LIN {X 0,Y 524.655,Z 657.487,A -85,B 0,C 180,E1 -4783.755,E2 -4783.755} C_VEL
LIN {X 0,Y 525.074,Z 645.522,A -85,B 0,C 180,E1 -4784.931,E2 -4784.931} C_VEL
LIN {X 0,Y 525.538,Z 633.607,A -85,B 0,C 180,E1 -4785.91,E2 -4785.91} C_VEL
LIN {X 0,Y 525.983,Z 620.728,A -85,B 0,C 180,E1 -4786.794,E2 -4786.794} C_VEL
LIN {X 0,Y 526.424,Z 606.681,A -85,B 0,C 180,E1 -4787.581,E2 -4787.581} C_VEL
LIN {X 0,Y 526.898,Z 592.222,A -85,B 0,C 180,E1 -4788.217,E2 -4788.217} C_VEL
LIN {X 0,Y 527.248,Z 577.139,A -85,B 0,C 180,E1 -4788.715,E2 -4788.715} C_VEL
LIN {X 0,Y 527.506,Z 562.381,A -85,B 0,C 180,E1 -4789.05,E2 -4789.05} C_VEL
LIN {X 0,Y 528.507,Z 412.087,A -85,B 0,C 180,E1 -4791.163,E2 -4791.163} C_VEL
LIN {X 0,Y 525.9,Z 396.895,A -85,B 0,C 180,E1 -4791.514,E2 -4791.514} C_VEL
LIN {X 0,Y 526.479,Z 374.491,A -85,B 0,C 180,E1 -4794.235,E2 -4794.235} C_VEL
LIN {X 0,Y 527.196,Z 352.396,A -85,B 0,C 180,E1 -4796.952,E2 -4796.952} C_VEL
LIN {X 0,Y 527.268,Z 349.014,A -85,B 0,C 180,E1 -4797.377,E2 -4797.377} C_VEL
LIN {X 0,Y 524.306,Z 336.37,A -85,B 0,C 180,E1 -4799.154,E2 -4799.154} C_VEL
LIN {X 0,Y 523.938,Z 334.849,A -85,B 0,C 180,E1 -4799.406,E2 -4799.406} C_VEL
LIN {X 0,Y 523.931,Z 334.844,A -85,B 0,C 180,E1 -4802.449,E2 -4802.449} C_VEL
LIN {X 0,Y 523.918,Z 334.851,A -85,B 0,C 180,E1 -4805.226,E2 -4805.226} C_VEL
LIN {X 0,Y 523.914,Z 334.848,A -85,B 0,C 180,E1 -4808.101,E2 -4808.101} C_VEL
LIN {X 0,Y 523.96,Z 334.847,A -85,B 0,C 180,E1 -4811.311,E2 -4811.311} C_VEL
LIN {X 0,Y 523.954,Z 334.841,A -85,B 0,C 180,E1 -4814.691,E2 -4814.691} C_VEL
LIN {X 0,Y 523.954,Z 334.84,A -85,B 0,C 180,E1 -4817.881,E2 -4817.881} C_VEL
LIN {X 0,Y 523.919,Z 334.848,A -85,B 0,C 180,E1 -4820.915,E2 -4820.915} C_VEL
LIN {X 0,Y 523.925,Z 334.843,A -85,B 0,C 180,E1 -4823.828,E2 -4823.828} C_VEL
LIN {X 0,Y 523.939,Z 334.843,A -85,B 0,C 180,E1 -4826.636,E2 -4826.636} C_VEL
LIN {X 0,Y 523.952,Z 334.844,A -85,B 0,C 180,E1 -4829.356,E2 -4829.356} C_VEL
LIN {X 0,Y 523.974,Z 334.836,A -85,B 0,C 180,E1 -4832.281,E2 -4832.281} C_VEL
LIN {X 0,Y 523.95,Z 334.841,A -85,B 0,C 180,E1 -4834.581,E2 -4834.581} C_VEL
LIN {X 0,Y 523.914,Z 334.853,A -85,B 0,C 180,E1 -4837.107,E2 -4837.107} C_VEL
LIN {X 0,Y 523.976,Z 334.836,A -85,B 0,C 180,E1 -4839.866,E2 -4839.866} C_VEL
LIN {X 0,Y 523.964,Z 334.844,A -85,B 0,C 180,E1 -4842.837,E2 -4842.837} C_VEL
LIN {X 0,Y 523.974,Z 334.842,A -85,B 0,C 180,E1 -4845.236,E2 -4845.236} C_VEL
LIN {X 0,Y 524.01,Z 334.833,A -85,B 0,C 180,E1 -4848.394,E2 -4848.394} C_VEL
LIN {X 0,Y 524.001,Z 334.835,A -85,B 0,C 180,E1 -4851.516,E2 -4851.516} C_VEL
LIN {X 0,Y 524.079,Z 334.827,A -85,B 0,C 180,E1 -4854.614,E2 -4854.614} C_VEL
LIN {X 0,Y 524.111,Z 334.82,A -85,B 0,C 180,E1 -4857.695,E2 -4857.695} C_VEL
LIN {X 0,Y 524.122,Z 334.825,A -85,B 0,C 180,E1 -4860.769,E2 -4860.769} C_VEL
LIN {X 0,Y 524.068,Z 334.831,A -85,B 0,C 180,E1 -4863.075,E2 -4863.075} C_VEL
LIN {X 0,Y 524.049,Z 334.828,A -85,B 0,C 180,E1 -4866.159,E2 -4866.159} C_VEL
LIN {X 0,Y 523.997,Z 334.836,A -85,B 0,C 180,E1 -4869.262,E2 -4869.262} C_VEL
LIN {X 0,Y 524.001,Z 334.833,A -85,B 0,C 180,E1 -4871.74,E2 -4871.74} C_VEL
LIN {X 0,Y 523.991,Z 334.839,A -85,B 0,C 180,E1 -4875.053,E2 -4875.053} C_VEL
LIN {X 0,Y 523.962,Z 334.838,A -85,B 0,C 180,E1 -4877.969,E2 -4877.969} C_VEL
LIN {X 0,Y 523.97,Z 334.841,A -85,B 0,C 180,E1 -4880.41,E2 -4880.41} C_VEL
LIN {X 0,Y 523.909,Z 334.851,A -85,B 0,C 180,E1 -4882.894,E2 -4882.894} C_VEL
LIN {X 0,Y 523.934,Z 334.842,A -85,B 0,C 180,E1 -4885.42,E2 -4885.42} C_VEL
LIN {X 0,Y 523.952,Z 334.84,A -85,B 0,C 180,E1 -4888,E2 -4888} C_VEL
LIN {X 0,Y 523.944,Z 334.847,A -85,B 0,C 180,E1 -4890.855,E2 -4890.855} C_VEL
LIN {X 0,Y 523.96,Z 334.838,A -85,B 0,C 180,E1 -4893.735,E2 -4893.735} C_VEL
LIN {X 0,Y 523.919,Z 334.849,A -85,B 0,C 180,E1 -4896.404,E2 -4896.404} C_VEL
LIN {X 0,Y 523.919,Z 334.846,A -85,B 0,C 180,E1 -4899.085,E2 -4899.085} C_VEL
LIN {X 0,Y 523.94,Z 334.843,A -85,B 0,C 180,E1 -4902.121,E2 -4902.121} C_VEL
LIN {X 0,Y 523.941,Z 334.841,A -85,B 0,C 180,E1 -4905.311,E2 -4905.311} C_VEL
LIN {X 0,Y 523.9,Z 334.849,A -85,B 0,C 180,E1 -4906.913,E2 -4906.913} C_VEL
LIN {X 0,Y 523.24,Z 334.929,A -85,B 0,C 180,E1 -4907.555,E2 -4907.555} C_VEL
LIN {X 0,Y 520.406,Z 335.29,A -85,B 0,C 180,E1 -4908.597,E2 -4908.597} C_VEL
LIN {X 0,Y 518.005,Z 335.589,A -85,B 0,C 180,E1 -4909.436,E2 -4909.436} C_VEL
LIN {X 0,Y 516.969,Z 335.715,A -85,B 0,C 180,E1 -4910.083,E2 -4910.083} C_VEL
LIN {X 0,Y 516.882,Z 335.725,A -85,B 0,C 180,E1 -4910.303,E2 -4910.303} C_VEL
LIN {X 0,Y 516.854,Z 335.723,A -85,B 0,C 180,E1 -4913.347,E2 -4913.347} C_VEL
LIN {X 0,Y 516.908,Z 335.72,A -85,B 0,C 180,E1 -4916.121,E2 -4916.121} C_VEL
LIN {X 0,Y 516.891,Z 335.721,A -85,B 0,C 180,E1 -4918.937,E2 -4918.937} C_VEL
LIN {X 0,Y 516.863,Z 335.722,A -85,B 0,C 180,E1 -4921.582,E2 -4921.582} C_VEL
LIN {X 0,Y 516.879,Z 335.725,A -85,B 0,C 180,E1 -4924.209,E2 -4924.209} C_VEL
LIN {X 0,Y 516.86,Z 335.726,A -85,B 0,C 180,E1 -4926.776,E2 -4926.776} C_VEL
LIN {X 0,Y 516.94,Z 335.713,A -85,B 0,C 180,E1 -4929.733,E2 -4929.733} C_VEL
LIN {X 0,Y 516.882,Z 335.726,A -85,B 0,C 180,E1 -4932.595,E2 -4932.595} C_VEL
LIN {X 0,Y 516.939,Z 335.714,A -85,B 0,C 180,E1 -4935.03,E2 -4935.03} C_VEL
LIN {X 0,Y 516.971,Z 335.716,A -85,B 0,C 180,E1 -4938.234,E2 -4938.234} C_VEL
LIN {X 0,Y 516.934,Z 335.713,A -85,B 0,C 180,E1 -4941.399,E2 -4941.399} C_VEL
LIN {X 0,Y 516.985,Z 335.712,A -85,B 0,C 180,E1 -4944.54,E2 -4944.54} C_VEL
LIN {X 0,Y 517.077,Z 335.697,A -85,B 0,C 180,E1 -4947.663,E2 -4947.663} C_VEL
LIN {X 0,Y 517.01,Z 335.706,A -85,B 0,C 180,E1 -4950.779,E2 -4950.779} C_VEL
LIN {X 0,Y 517.076,Z 335.703,A -85,B 0,C 180,E1 -4952.337,E2 -4952.337} C_VEL
LIN {X 0,Y 516.975,Z 335.717,A -85,B 0,C 180,E1 -4956.244,E2 -4956.244} C_VEL
LIN {X 0,Y 516.911,Z 335.716,A -85,B 0,C 180,E1 -4959.39,E2 -4959.39} C_VEL
LIN {X 0,Y 516.902,Z 335.722,A -85,B 0,C 180,E1 -4962.565,E2 -4962.565} C_VEL
LIN {X 0,Y 516.832,Z 335.733,A -85,B 0,C 180,E1 -4965.782,E2 -4965.782} C_VEL
LIN {X 0,Y 516.878,Z 335.791,A -85,B 0,C 180,E1 -4967.049,E2 -4967.049} C_VEL
LIN {X 0,Y 518.301,Z 342.495,A -85,B 0,C 180,E1 -4968.249,E2 -4968.249} C_VEL
LIN {X 0,Y 520.55,Z 349.737,A -85,B 0,C 180,E1 -4968.46,E2 -4968.46} C_VEL
LIN {X 0,Y 521.981,Z 356.506,A -85,B 0,C 180,E1 -4968.624,E2 -4968.624} C_VEL
LIN {X 0,Y 520.841,Z 507.169,A -85,B 0,C 180,E1 -4970.79,E2 -4970.79} C_VEL
LIN {X 0,Y 520.577,Z 522.264,A -85,B 0,C 180,E1 -4971.165,E2 -4971.165} C_VEL
LIN {X 0,Y 520.179,Z 537.472,A -85,B 0,C 180,E1 -4971.707,E2 -4971.707} C_VEL
LIN {X 0,Y 519.763,Z 552.073,A -85,B 0,C 180,E1 -4972.403,E2 -4972.403} C_VEL
LIN {X 0,Y 519.251,Z 565.638,A -85,B 0,C 180,E1 -4973.217,E2 -4973.217} C_VEL
LIN {X 0,Y 518.701,Z 578.837,A -85,B 0,C 180,E1 -4974.189,E2 -4974.189} C_VEL
LIN {X 0,Y 518.145,Z 591.198,A -85,B 0,C 180,E1 -4975.294,E2 -4975.294} C_VEL
LIN {X 0,Y 517.709,Z 601.985,A -85,B 0,C 180,E1 -4976.451,E2 -4976.451} C_VEL
LIN {X 0,Y 517.308,Z 612.091,A -85,B 0,C 180,E1 -4977.74,E2 -4977.74} C_VEL
LIN {X 0,Y 516.968,Z 620.889,A -85,B 0,C 180,E1 -4979.079,E2 -4979.079} C_VEL
LIN {X 0,Y 516.683,Z 629.217,A -85,B 0,C 180,E1 -4980.61,E2 -4980.61} C_VEL
LIN {X 0,Y 516.497,Z 635.604,A -85,B 0,C 180,E1 -4982.051,E2 -4982.051} C_VEL
LIN {X 0,Y 516.368,Z 640.556,A -85,B 0,C 180,E1 -4983.426,E2 -4983.426} C_VEL
LIN {X 0,Y 516.253,Z 644.668,A -85,B 0,C 180,E1 -4984.874,E2 -4984.874} C_VEL
LIN {X 0,Y 516.177,Z 648.074,A -85,B 0,C 180,E1 -4986.552,E2 -4986.552} C_VEL
LIN {X 0,Y 516.14,Z 649.735,A -85,B 0,C 180,E1 -4987.837,E2 -4987.837} C_VEL
LIN {X 0,Y 516.152,Z 650.678,A -85,B 0,C 180,E1 -4989.093,E2 -4989.093} C_VEL
LIN {X 0,Y 516.173,Z 650.75,A -85,B 0,C 180,E1 -4990.81,E2 -4990.81} C_VEL
LIN {X 0,Y 516.166,Z 650.148,A -85,B 0,C 180,E1 -4991.85,E2 -4991.85} C_VEL
LIN {X 0,Y 516.175,Z 648.994,A -85,B 0,C 180,E1 -4992.905,E2 -4992.905} C_VEL
LIN {X 0,Y 516.288,Z 646.397,A -85,B 0,C 180,E1 -4994.453,E2 -4994.453} C_VEL
LIN {X 0,Y 516.383,Z 642.122,A -85,B 0,C 180,E1 -4996.165,E2 -4996.165} C_VEL
LIN {X 0,Y 516.442,Z 636.865,A -85,B 0,C 180,E1 -4997.735,E2 -4997.735} C_VEL
LIN {X 0,Y 516.635,Z 630.492,A -85,B 0,C 180,E1 -4999.234,E2 -4999.234} C_VEL
LIN {X 0,Y 516.904,Z 622.228,A -85,B 0,C 180,E1 -5000.805,E2 -5000.805} C_VEL
LIN {X 0,Y 517.25,Z 613.537,A -85,B 0,C 180,E1 -5002.161,E2 -5002.161} C_VEL
LIN {X 0,Y 517.705,Z 602.748,A -85,B 0,C 180,E1 -5003.564,E2 -5003.564} C_VEL
LIN {X 0,Y 518.226,Z 591.212,A -85,B 0,C 180,E1 -5004.804,E2 -5004.804} C_VEL
LIN {X 0,Y 518.709,Z 578.953,A -85,B 0,C 180,E1 -5005.902,E2 -5005.902} C_VEL
LIN {X 0,Y 519.183,Z 566.64,A -85,B 0,C 180,E1 -5006.818,E2 -5006.818} C_VEL
LIN {X 0,Y 519.754,Z 552.758,A -85,B 0,C 180,E1 -5007.659,E2 -5007.659} C_VEL
LIN {X 0,Y 520.167,Z 538.55,A -85,B 0,C 180,E1 -5008.342,E2 -5008.342} C_VEL
LIN {X 0,Y 520.558,Z 522.971,A -85,B 0,C 180,E1 -5008.908,E2 -5008.908} C_VEL
LIN {X 0,Y 520.81,Z 507.957,A -85,B 0,C 180,E1 -5009.285,E2 -5009.285} C_VEL
LIN {X 0,Y 521.407,Z 427.366,A -85,B 0,C 180,E1 -5010.459,E2 -5010.459} C_VEL
LIN {X 0,Y 521.907,Z 355.675,A -85,B 0,C 180,E1 -5011.489,E2 -5011.489} C_VEL
LIN {X 0,Y 519.249,Z 345.342,A -85,B 0,C 180,E1 -5011.761,E2 -5011.761} C_VEL
LIN {X 0,Y 518.421,Z 342.909,A -85,B 0,C 180,E1 -5011.862,E2 -5011.862} C_VEL
LIN {X 0,Y 516.883,Z 335.728,A -85,B 0,C 180,E1 -5013.203,E2 -5013.203} C_VEL
LIN {X 0,Y 516.871,Z 335.729,A -85,B 0,C 180,E1 -5015.926,E2 -5015.926} C_VEL
LIN {X 0,Y 516.867,Z 335.724,A -85,B 0,C 180,E1 -5018.461,E2 -5018.461} C_VEL
LIN {X 0,Y 516.882,Z 335.721,A -85,B 0,C 180,E1 -5020.954,E2 -5020.954} C_VEL
LIN {X 0,Y 516.844,Z 335.728,A -85,B 0,C 180,E1 -5023.408,E2 -5023.408} C_VEL
LIN {X 0,Y 516.884,Z 335.728,A -85,B 0,C 180,E1 -5025.833,E2 -5025.833} C_VEL
LIN {X 0,Y 516.95,Z 335.714,A -85,B 0,C 180,E1 -5029.028,E2 -5029.028} C_VEL
LIN {X 0,Y 516.926,Z 335.717,A -85,B 0,C 180,E1 -5032.186,E2 -5032.186} C_VEL
LIN {X 0,Y 516.989,Z 335.707,A -85,B 0,C 180,E1 -5034.539,E2 -5034.539} C_VEL
LIN {X 0,Y 517.078,Z 335.704,A -85,B 0,C 180,E1 -5037.663,E2 -5037.663} C_VEL
LIN {X 0,Y 517.088,Z 335.698,A -85,B 0,C 180,E1 -5040,E2 -5040} C_VEL
LIN {X 0,Y 517.082,Z 335.696,A -85,B 0,C 180,E1 -5042.337,E2 -5042.337} C_VEL
LIN {X 0,Y 517.015,Z 335.711,A -85,B 0,C 180,E1 -5045.46,E2 -5045.46} C_VEL
LIN {X 0,Y 516.957,Z 335.712,A -85,B 0,C 180,E1 -5048.6,E2 -5048.6} C_VEL
LIN {X 0,Y 516.955,Z 335.714,A -85,B 0,C 180,E1 -5051.807,E2 -5051.807} C_VEL
LIN {X 0,Y 516.946,Z 335.719,A -85,B 0,C 180,E1 -5055.146,E2 -5055.146} C_VEL
LIN {X 0,Y 516.918,Z 335.715,A -85,B 0,C 180,E1 -5058.222,E2 -5058.222} C_VEL
LIN {X 0,Y 516.914,Z 335.718,A -85,B 0,C 180,E1 -5060.701,E2 -5060.701} C_VEL
LIN {X 0,Y 516.893,Z 335.718,A -85,B 0,C 180,E1 -5064.073,E2 -5064.073} C_VEL
LIN {X 0,Y 516.926,Z 335.717,A -85,B 0,C 180,E1 -5066.657,E2 -5066.657} C_VEL
LIN {X 0,Y 516.913,Z 335.719,A -85,B 0,C 180,E1 -5069.523,E2 -5069.523} C_VEL
LIN {X 0,Y 516.897,Z 335.72,A -85,B 0,C 180,E1 -5072.543,E2 -5072.543} C_VEL
LIN {X 0,Y 516.868,Z 335.728,A -85,B 0,C 180,E1 -5075.329,E2 -5075.329} C_VEL
LIN {X 0,Y 516.882,Z 335.722,A -85,B 0,C 180,E1 -5077.943,E2 -5077.943} C_VEL
LIN {X 0,Y 516.887,Z 335.727,A -85,B 0,C 180,E1 -5080.741,E2 -5080.741} C_VEL
LIN {X 0,Y 516.886,Z 335.728,A -85,B 0,C 180,E1 -5082.831,E2 -5082.831} C_VEL
LIN {X 0,Y 516.924,Z 335.723,A -85,B 0,C 180,E1 -5085.01,E2 -5085.01} C_VEL
LIN {X 0,Y 516.917,Z 335.72,A -85,B 0,C 180,E1 -5088.398,E2 -5088.398} C_VEL
LIN {X 0,Y 516.883,Z 335.725,A -85,B 0,C 180,E1 -5091.284,E2 -5091.284} C_VEL
LIN {X 0,Y 516.872,Z 335.725,A -85,B 0,C 180,E1 -5094.219,E2 -5094.219} C_VEL
LIN {X 0,Y 516.896,Z 335.727,A -85,B 0,C 180,E1 -5097.053,E2 -5097.053} C_VEL
LIN {X 0,Y 516.911,Z 335.725,A -85,B 0,C 180,E1 -5100.364,E2 -5100.364} C_VEL
LIN {X 0,Y 516.91,Z 335.805,A -85,B 0,C 180,E1 -5100.476,E2 -5100.476} C_VEL
LIN {X 0,Y 520.193,Z 349.607,A -85,B 0,C 180,E1 -5102.436,E2 -5102.436} C_VEL
LIN {X 0,Y 519.867,Z 364.959,A -85,B 0,C 180,E1 -5104.367,E2 -5104.367} C_VEL
LIN {X 0,Y 519.106,Z 389.232,A -85,B 0,C 180,E1 -5107.356,E2 -5107.356} C_VEL
LIN {X 0,Y 518.953,Z 396.135,A -85,B 0,C 180,E1 -5108.199,E2 -5108.199} C_VEL
LIN {X 0,Y 521.84,Z 413.333,A -85,B 0,C 180,E1 -5108.583,E2 -5108.583} C_VEL
LIN {X 0,Y 520.752,Z 563.435,A -85,B 0,C 180,E1 -5110.732,E2 -5110.732} C_VEL
LIN {X 0,Y 520.451,Z 578.968,A -85,B 0,C 180,E1 -5111.111,E2 -5111.111} C_VEL
LIN {X 0,Y 520.044,Z 593.948,A -85,B 0,C 180,E1 -5111.636,E2 -5111.636} C_VEL
LIN {X 0,Y 519.555,Z 607.913,A -85,B 0,C 180,E1 -5112.28,E2 -5112.28} C_VEL
LIN {X 0,Y 519.025,Z 621.616,A -85,B 0,C 180,E1 -5113.074,E2 -5113.074} C_VEL
LIN {X 0,Y 518.525,Z 635.554,A -85,B 0,C 180,E1 -5114.07,E2 -5114.07} C_VEL
LIN {X 0,Y 517.98,Z 648.16,A -85,B 0,C 180,E1 -5115.161,E2 -5115.161} C_VEL
LIN {X 0,Y 517.585,Z 658.732,A -85,B 0,C 180,E1 -5116.253,E2 -5116.253} C_VEL
LIN {X 0,Y 517.214,Z 668.547,A -85,B 0,C 180,E1 -5117.443,E2 -5117.443} C_VEL
LIN {X 0,Y 516.923,Z 678.187,A -85,B 0,C 180,E1 -5118.829,E2 -5118.829} C_VEL
LIN {X 0,Y 516.625,Z 686.213,A -85,B 0,C 180,E1 -5120.209,E2 -5120.209} C_VEL
LIN {X 0,Y 516.479,Z 693.711,A -85,B 0,C 180,E1 -5121.785,E2 -5121.785} C_VEL
LIN {X 0,Y 516.391,Z 698.314,A -85,B 0,C 180,E1 -5122.964,E2 -5122.964} C_VEL
LIN {X 0,Y 516.352,Z 703.191,A -85,B 0,C 180,E1 -5124.532,E2 -5124.532} C_VEL
LIN {X 0,Y 516.293,Z 706.761,A -85,B 0,C 180,E1 -5126.097,E2 -5126.097} C_VEL
LIN {X 0,Y 516.258,Z 709.108,A -85,B 0,C 180,E1 -5127.659,E2 -5127.659} C_VEL
LIN {X 0,Y 516.156,Z 710.284,A -85,B 0,C 180,E1 -5129.219,E2 -5129.219} C_VEL
LIN {X 0,Y 516.156,Z 710.283,A -85,B 0,C 180,E1 -5130.78,E2 -5130.78} C_VEL
LIN {X 0,Y 516.258,Z 709.105,A -85,B 0,C 180,E1 -5132.34,E2 -5132.34} C_VEL
LIN {X 0,Y 516.293,Z 706.76,A -85,B 0,C 180,E1 -5133.902,E2 -5133.902} C_VEL
LIN {X 0,Y 516.351,Z 703.201,A -85,B 0,C 180,E1 -5135.467,E2 -5135.467} C_VEL
LIN {X 0,Y 516.391,Z 698.336,A -85,B 0,C 180,E1 -5137.035,E2 -5137.035} C_VEL
LIN {X 0,Y 516.54,Z 692.038,A -85,B 0,C 180,E1 -5138.607,E2 -5138.607} C_VEL
LIN {X 0,Y 516.727,Z 684.128,A -85,B 0,C 180,E1 -5140.184,E2 -5140.184} C_VEL
LIN {X 0,Y 516.959,Z 675.716,A -85,B 0,C 180,E1 -5141.567,E2 -5141.567} C_VEL
LIN {X 0,Y 517.348,Z 665.588,A -85,B 0,C 180,E1 -5142.952,E2 -5142.952} C_VEL
LIN {X 0,Y 517.704,Z 655.236,A -85,B 0,C 180,E1 -5144.143,E2 -5144.143} C_VEL
LIN {X 0,Y 518.205,Z 643.267,A -85,B 0,C 180,E1 -5145.301,E2 -5145.301} C_VEL
LIN {X 0,Y 518.727,Z 630.524,A -85,B 0,C 180,E1 -5146.327,E2 -5146.327} C_VEL
LIN {X 0,Y 519.241,Z 617.051,A -85,B 0,C 180,E1 -5147.222,E2 -5147.222} C_VEL
LIN {X 0,Y 519.773,Z 602.179,A -85,B 0,C 180,E1 -5148.017,E2 -5148.017} C_VEL
LIN {X 0,Y 520.232,Z 587.764,A -85,B 0,C 180,E1 -5148.612,E2 -5148.612} C_VEL
LIN {X 0,Y 520.546,Z 573.066,A -85,B 0,C 180,E1 -5149.062,E2 -5149.062} C_VEL
LIN {X 0,Y 520.844,Z 558.221,A -85,B 0,C 180,E1 -5149.362,E2 -5149.362} C_VEL
LIN {X 0,Y 521.83,Z 412.162,A -85,B 0,C 180,E1 -5151.44,E2 -5151.44} C_VEL
LIN {X 0,Y 519.009,Z 396.667,A -85,B 0,C 180,E1 -5151.795,E2 -5151.795} C_VEL
LIN {X 0,Y 519.607,Z 375.836,A -85,B 0,C 180,E1 -5154.364,E2 -5154.364} C_VEL
LIN {X 0,Y 520.362,Z 355.067,A -85,B 0,C 180,E1 -5156.951,E2 -5156.951} C_VEL
LIN {X 0,Y 520.403,Z 350.385,A -85,B 0,C 180,E1 -5157.551,E2 -5157.551} C_VEL
LIN {X 0,Y 516.913,Z 335.723,A -85,B 0,C 180,E1 -5159.656,E2 -5159.656} C_VEL
LIN {X 0,Y 516.893,Z 335.724,A -85,B 0,C 180,E1 -5162.947,E2 -5162.947} C_VEL
LIN {X 0,Y 516.869,Z 335.727,A -85,B 0,C 180,E1 -5165.78,E2 -5165.78} C_VEL
LIN {X 0,Y 516.88,Z 335.726,A -85,B 0,C 180,E1 -5168.715,E2 -5168.715} C_VEL
LIN {X 0,Y 516.914,Z 335.718,A -85,B 0,C 180,E1 -5171.774,E2 -5171.774} C_VEL
LIN {X 0,Y 516.92,Z 335.721,A -85,B 0,C 180,E1 -5175.01,E2 -5175.01} C_VEL
LIN {X 0,Y 516.915,Z 335.716,A -85,B 0,C 180,E1 -5178.398,E2 -5178.398} C_VEL
LIN {X 0,Y 516.879,Z 335.728,A -85,B 0,C 180,E1 -5181.284,E2 -5181.284} C_VEL
LIN {X 0,Y 516.888,Z 335.719,A -85,B 0,C 180,E1 -5184.221,E2 -5184.221} C_VEL
LIN {X 0,Y 516.892,Z 335.726,A -85,B 0,C 180,E1 -5187.053,E2 -5187.053} C_VEL
LIN {X 0,Y 516.889,Z 335.72,A -85,B 0,C 180,E1 -5189.796,E2 -5189.796} C_VEL
LIN {X 0,Y 516.923,Z 335.716,A -85,B 0,C 180,E1 -5192.467,E2 -5192.467} C_VEL
LIN {X 0,Y 516.908,Z 335.726,A -85,B 0,C 180,E1 -5195.072,E2 -5195.072} C_VEL
LIN {X 0,Y 516.867,Z 335.723,A -85,B 0,C 180,E1 -5197.622,E2 -5197.622} C_VEL
LIN {X 0,Y 516.929,Z 335.714,A -85,B 0,C 180,E1 -5200.13,E2 -5200.13} C_VEL
LIN {X 0,Y 516.926,Z 335.717,A -85,B 0,C 180,E1 -5202.596,E2 -5202.596} C_VEL
LIN {X 0,Y 516.94,Z 335.722,A -85,B 0,C 180,E1 -5205.03,E2 -5205.03} C_VEL
LIN {X 0,Y 516.963,Z 335.71,A -85,B 0,C 180,E1 -5208.234,E2 -5208.234} C_VEL
LIN {X 0,Y 516.966,Z 335.712,A -85,B 0,C 180,E1 -5211.4,E2 -5211.4} C_VEL
LIN {X 0,Y 517,Z 335.705,A -85,B 0,C 180,E1 -5213.757,E2 -5213.757} C_VEL
LIN {X 0,Y 517.011,Z 335.712,A -85,B 0,C 180,E1 -5216.883,E2 -5216.883} C_VEL
LIN {X 0,Y 517.084,Z 335.695,A -85,B 0,C 180,E1 -5220,E2 -5220} C_VEL
LIN {X 0,Y 517.009,Z 335.709,A -85,B 0,C 180,E1 -5223.117,E2 -5223.117} C_VEL
LIN {X 0,Y 517.013,Z 335.705,A -85,B 0,C 180,E1 -5226.243,E2 -5226.243} C_VEL
LIN {X 0,Y 516.951,Z 335.713,A -85,B 0,C 180,E1 -5229.39,E2 -5229.39} C_VEL
LIN {X 0,Y 516.95,Z 335.711,A -85,B 0,C 180,E1 -5231.808,E2 -5231.808} C_VEL
LIN {X 0,Y 516.943,Z 335.716,A -85,B 0,C 180,E1 -5235.147,E2 -5235.147} C_VEL
LIN {X 0,Y 516.923,Z 335.716,A -85,B 0,C 180,E1 -5238.223,E2 -5238.223} C_VEL
LIN {X 0,Y 516.911,Z 335.725,A -85,B 0,C 180,E1 -5240.702,E2 -5240.702} C_VEL
LIN {X 0,Y 516.901,Z 335.718,A -85,B 0,C 180,E1 -5244.073,E2 -5244.073} C_VEL
LIN {X 0,Y 516.903,Z 335.726,A -85,B 0,C 180,E1 -5246.659,E2 -5246.659} C_VEL
LIN {X 0,Y 516.91,Z 335.716,A -85,B 0,C 180,E1 -5249.524,E2 -5249.524} C_VEL
LIN {X 0,Y 516.894,Z 335.725,A -85,B 0,C 180,E1 -5252.544,E2 -5252.544} C_VEL
LIN {X 0,Y 516.879,Z 335.721,A -85,B 0,C 180,E1 -5255.332,E2 -5255.332} C_VEL
LIN {X 0,Y 516.88,Z 335.721,A -85,B 0,C 180,E1 -5257.944,E2 -5257.944} C_VEL
LIN {X 0,Y 516.881,Z 335.727,A -85,B 0,C 180,E1 -5260.742,E2 -5260.742} C_VEL
LIN {X 0,Y 516.881,Z 335.721,A -85,B 0,C 180,E1 -5263.904,E2 -5263.904} C_VEL
LIN {X 0,Y 516.849,Z 335.724,A -85,B 0,C 180,E1 -5266.915,E2 -5266.915} C_VEL
LIN {X 0,Y 516.885,Z 335.719,A -85,B 0,C 180,E1 -5269.59,E2 -5269.59} C_VEL
LIN {X 0,Y 516.882,Z 335.725,A -85,B 0,C 180,E1 -5270.303,E2 -5270.303} C_VEL
LIN {X 0,Y 516.207,Z 335.808,A -85,B 0,C 180,E1 -5270.953,E2 -5270.953} C_VEL
LIN {X 0,Y 513.348,Z 336.162,A -85,B 0,C 180,E1 -5272.008,E2 -5272.008} C_VEL
LIN {X 0,Y 510.934,Z 336.465,A -85,B 0,C 180,E1 -5272.859,E2 -5272.859} C_VEL
LIN {X 0,Y 509.894,Z 336.591,A -85,B 0,C 180,E1 -5273.515,E2 -5273.515} C_VEL
LIN {X 0,Y 509.807,Z 336.601,A -85,B 0,C 180,E1 -5273.737,E2 -5273.737} C_VEL
LIN {X 0,Y 509.86,Z 336.603,A -85,B 0,C 180,E1 -5276.54,E2 -5276.54} C_VEL
LIN {X 0,Y 509.844,Z 336.596,A -85,B 0,C 180,E1 -5279.335,E2 -5279.335} C_VEL
LIN {X 0,Y 509.848,Z 336.599,A -85,B 0,C 180,E1 -5282.052,E2 -5282.052} C_VEL
LIN {X 0,Y 509.808,Z 336.606,A -85,B 0,C 180,E1 -5284.701,E2 -5284.701} C_VEL
LIN {X 0,Y 509.828,Z 336.598,A -85,B 0,C 180,E1 -5287.459,E2 -5287.459} C_VEL
LIN {X 0,Y 509.918,Z 336.589,A -85,B 0,C 180,E1 -5289.845,E2 -5289.845} C_VEL
LIN {X 0,Y 509.855,Z 336.604,A -85,B 0,C 180,E1 -5292.347,E2 -5292.347} C_VEL
LIN {X 0,Y 509.889,Z 336.594,A -85,B 0,C 180,E1 -5294.819,E2 -5294.819} C_VEL
LIN {X 0,Y 509.905,Z 336.594,A -85,B 0,C 180,E1 -5298.125,E2 -5298.125} C_VEL
LIN {X 0,Y 509.888,Z 336.591,A -85,B 0,C 180,E1 -5301.28,E2 -5301.28} C_VEL
LIN {X 0,Y 509.92,Z 336.588,A -85,B 0,C 180,E1 -5303.67,E2 -5303.67} C_VEL
LIN {X 0,Y 509.892,Z 336.592,A -85,B 0,C 180,E1 -5306.84,E2 -5306.84} C_VEL
LIN {X 0,Y 509.929,Z 336.593,A -85,B 0,C 180,E1 -5308.421,E2 -5308.421} C_VEL
LIN {X 0,Y 509.963,Z 336.583,A -85,B 0,C 180,E1 -5310.79,E2 -5310.79} C_VEL
LIN {X 0,Y 510.045,Z 336.579,A -85,B 0,C 180,E1 -5312.369,E2 -5312.369} C_VEL
LIN {X 0,Y 509.941,Z 336.585,A -85,B 0,C 180,E1 -5315.536,E2 -5315.536} C_VEL
LIN {X 0,Y 509.879,Z 336.597,A -85,B 0,C 180,E1 -5317.923,E2 -5317.923} C_VEL
LIN {X 0,Y 509.865,Z 336.595,A -85,B 0,C 180,E1 -5321.127,E2 -5321.127} C_VEL
LIN {X 0,Y 509.824,Z 336.603,A -85,B 0,C 180,E1 -5323.553,E2 -5323.553} C_VEL
LIN {X 0,Y 509.793,Z 336.612,A -85,B 0,C 180,E1 -5326.005,E2 -5326.005} C_VEL
LIN {X 0,Y 509.838,Z 336.796,A -85,B 0,C 180,E1 -5326.827,E2 -5326.827} C_VEL
LIN {X 0,Y 511.145,Z 342.787,A -85,B 0,C 180,E1 -5327.918,E2 -5327.918} C_VEL
LIN {X 0,Y 513.814,Z 350.508,A -85,B 0,C 180,E1 -5328.169,E2 -5328.169} C_VEL
LIN {X 0,Y 515.379,Z 358.221,A -85,B 0,C 180,E1 -5328.356,E2 -5328.356} C_VEL
LIN {X 0,Y 514.162,Z 507.222,A -85,B 0,C 180,E1 -5330.53,E2 -5330.53} C_VEL
LIN {X 0,Y 513.847,Z 522.474,A -85,B 0,C 180,E1 -5330.909,E2 -5330.909} C_VEL
LIN {X 0,Y 513.477,Z 537.513,A -85,B 0,C 180,E1 -5331.451,E2 -5331.451} C_VEL
LIN {X 0,Y 513.011,Z 551.765,A -85,B 0,C 180,E1 -5332.132,E2 -5332.132} C_VEL
LIN {X 0,Y 512.483,Z 564.759,A -85,B 0,C 180,E1 -5332.91,E2 -5332.91} C_VEL
LIN {X 0,Y 511.942,Z 576.774,A -85,B 0,C 180,E1 -5333.783,E2 -5333.783} C_VEL
LIN {X 0,Y 511.371,Z 589.483,A -85,B 0,C 180,E1 -5334.896,E2 -5334.896} C_VEL
LIN {X 0,Y 510.837,Z 601.08,A -85,B 0,C 180,E1 -5336.12,E2 -5336.12} C_VEL
LIN {X 0,Y 510.368,Z 611.74,A -85,B 0,C 180,E1 -5337.472,E2 -5337.472} C_VEL
LIN {X 0,Y 510.001,Z 620.711,A -85,B 0,C 180,E1 -5338.837,E2 -5338.837} C_VEL
LIN {X 0,Y 509.705,Z 628.301,A -85,B 0,C 180,E1 -5340.217,E2 -5340.217} C_VEL
LIN {X 0,Y 509.516,Z 634.674,A -85,B 0,C 180,E1 -5341.612,E2 -5341.612} C_VEL
LIN {X 0,Y 509.333,Z 640.077,A -85,B 0,C 180,E1 -5343.06,E2 -5343.06} C_VEL
LIN {X 0,Y 509.251,Z 644.169,A -85,B 0,C 180,E1 -5344.46,E2 -5344.46} C_VEL
LIN {X 0,Y 509.138,Z 646.543,A -85,B 0,C 180,E1 -5345.469,E2 -5345.469} C_VEL
LIN {X 0,Y 509.086,Z 648.906,A -85,B 0,C 180,E1 -5346.802,E2 -5346.802} C_VEL
LIN {X 0,Y 509.06,Z 650.685,A -85,B 0,C 180,E1 -5348.409,E2 -5348.409} C_VEL
LIN {X 0,Y 509.072,Z 651.188,A -85,B 0,C 180,E1 -5349.424,E2 -5349.424} C_VEL
LIN {X 0,Y 509.073,Z 651.202,A -85,B 0,C 180,E1 -5350.597,E2 -5350.597} C_VEL
LIN {X 0,Y 509.078,Z 650.626,A -85,B 0,C 180,E1 -5351.798,E2 -5351.798} C_VEL
LIN {X 0,Y 509.145,Z 648.403,A -85,B 0,C 180,E1 -5353.644,E2 -5353.644} C_VEL
LIN {X 0,Y 509.271,Z 645.148,A -85,B 0,C 180,E1 -5355.266,E2 -5355.266} C_VEL
LIN {X 0,Y 509.365,Z 640.253,A -85,B 0,C 180,E1 -5356.993,E2 -5356.993} C_VEL
LIN {X 0,Y 509.494,Z 634.517,A -85,B 0,C 180,E1 -5358.538,E2 -5358.538} C_VEL
LIN {X 0,Y 509.743,Z 627.247,A -85,B 0,C 180,E1 -5360.104,E2 -5360.104} C_VEL
LIN {X 0,Y 510.064,Z 619.759,A -85,B 0,C 180,E1 -5361.428,E2 -5361.428} C_VEL
LIN {X 0,Y 510.462,Z 609.903,A -85,B 0,C 180,E1 -5362.888,E2 -5362.888} C_VEL
LIN {X 0,Y 510.876,Z 600.772,A -85,B 0,C 180,E1 -5364.022,E2 -5364.022} C_VEL
LIN {X 0,Y 511.458,Z 588.772,A -85,B 0,C 180,E1 -5365.276,E2 -5365.276} C_VEL
LIN {X 0,Y 511.962,Z 576.532,A -85,B 0,C 180,E1 -5366.34,E2 -5366.34} C_VEL
LIN {X 0,Y 512.558,Z 562.745,A -85,B 0,C 180,E1 -5367.323,E2 -5367.323} C_VEL
LIN {X 0,Y 513.13,Z 548.772,A -85,B 0,C 180,E1 -5368.122,E2 -5368.122} C_VEL
LIN {X 0,Y 513.542,Z 534.243,A -85,B 0,C 180,E1 -5368.776,E2 -5368.776} C_VEL
LIN {X 0,Y 513.908,Z 518.92,A -85,B 0,C 180,E1 -5369.285,E2 -5369.285} C_VEL
LIN {X 0,Y 514.185,Z 503.013,A -85,B 0,C 180,E1 -5369.634,E2 -5369.634} C_VEL
LIN {X 0,Y 515.32,Z 356.831,A -85,B 0,C 180,E1 -5371.766,E2 -5371.766} C_VEL
LIN {X 0,Y 512.913,Z 347.688,A -85,B 0,C 180,E1 -5372.013,E2 -5372.013} C_VEL
LIN {X 0,Y 511.326,Z 343.478,A -85,B 0,C 180,E1 -5372.167,E2 -5372.167} C_VEL
LIN {X 0,Y 509.815,Z 336.607,A -85,B 0,C 180,E1 -5373.468,E2 -5373.468} C_VEL
LIN {X 0,Y 509.811,Z 336.607,A -85,B 0,C 180,E1 -5376.435,E2 -5376.435} C_VEL
LIN {X 0,Y 509.892,Z 336.599,A -85,B 0,C 180,E1 -5379.843,E2 -5379.843} C_VEL
LIN {X 0,Y 509.855,Z 336.597,A -85,B 0,C 180,E1 -5382.346,E2 -5382.346} C_VEL
LIN {X 0,Y 509.889,Z 336.593,A -85,B 0,C 180,E1 -5384.818,E2 -5384.818} C_VEL
LIN {X 0,Y 509.905,Z 336.594,A -85,B 0,C 180,E1 -5388.124,E2 -5388.124} C_VEL
LIN {X 0,Y 509.887,Z 336.596,A -85,B 0,C 180,E1 -5391.279,E2 -5391.279} C_VEL
LIN {X 0,Y 509.943,Z 336.585,A -85,B 0,C 180,E1 -5394.464,E2 -5394.464} C_VEL
LIN {X 0,Y 510.046,Z 336.579,A -85,B 0,C 180,E1 -5397.631,E2 -5397.631} C_VEL
LIN {X 0,Y 510.059,Z 336.574,A -85,B 0,C 180,E1 -5400,E2 -5400} C_VEL
LIN {X 0,Y 510.052,Z 336.571,A -85,B 0,C 180,E1 -5402.369,E2 -5402.369} C_VEL
LIN {X 0,Y 509.966,Z 336.59,A -85,B 0,C 180,E1 -5405.536,E2 -5405.536} C_VEL
LIN {X 0,Y 509.905,Z 336.591,A -85,B 0,C 180,E1 -5408.72,E2 -5408.72} C_VEL
LIN {X 0,Y 509.907,Z 336.591,A -85,B 0,C 180,E1 -5411.931,E2 -5411.931} C_VEL
LIN {X 0,Y 509.897,Z 336.597,A -85,B 0,C 180,E1 -5415.241,E2 -5415.241} C_VEL
LIN {X 0,Y 509.864,Z 336.594,A -85,B 0,C 180,E1 -5418.483,E2 -5418.483} C_VEL
LIN {X 0,Y 509.852,Z 336.602,A -85,B 0,C 180,E1 -5421.001,E2 -5421.001} C_VEL
LIN {X 0,Y 509.857,Z 336.595,A -85,B 0,C 180,E1 -5424.426,E2 -5424.426} C_VEL
LIN {X 0,Y 509.886,Z 336.598,A -85,B 0,C 180,E1 -5427.055,E2 -5427.055} C_VEL
LIN {X 0,Y 509.859,Z 336.596,A -85,B 0,C 180,E1 -5429.751,E2 -5429.751} C_VEL
LIN {X 0,Y 509.875,Z 336.597,A -85,B 0,C 180,E1 -5432.774,E2 -5432.774} C_VEL
LIN {X 0,Y 509.827,Z 336.603,A -85,B 0,C 180,E1 -5435.578,E2 -5435.578} C_VEL
LIN {X 0,Y 509.852,Z 336.599,A -85,B 0,C 180,E1 -5438.338,E2 -5438.338} C_VEL
LIN {X 0,Y 509.859,Z 336.599,A -85,B 0,C 180,E1 -5441.425,E2 -5441.425} C_VEL
LIN {X 0,Y 509.858,Z 336.602,A -85,B 0,C 180,E1 -5444.668,E2 -5444.668} C_VEL
LIN {X 0,Y 509.861,Z 336.597,A -85,B 0,C 180,E1 -5448.103,E2 -5448.103} C_VEL
LIN {X 0,Y 509.848,Z 336.604,A -85,B 0,C 180,E1 -5450.647,E2 -5450.647} C_VEL
LIN {X 0,Y 509.826,Z 336.602,A -85,B 0,C 180,E1 -5453.647,E2 -5453.647} C_VEL
LIN {X 0,Y 509.86,Z 336.602,A -85,B 0,C 180,E1 -5456.539,E2 -5456.539} C_VEL
LIN {X 0,Y 509.863,Z 336.601,A -85,B 0,C 180,E1 -5459.793,E2 -5459.793} C_VEL
LIN {X 0,Y 509.877,Z 336.631,A -85,B 0,C 180,E1 -5460.193,E2 -5460.193} C_VEL
LIN {X 0,Y 513.267,Z 350.876,A -85,B 0,C 180,E1 -5462.254,E2 -5462.254} C_VEL
LIN {X 0,Y 513.318,Z 357.705,A -85,B 0,C 180,E1 -5463.14,E2 -5463.14} C_VEL
LIN {X 0,Y 512.514,Z 381.522,A -85,B 0,C 180,E1 -5466.138,E2 -5466.138} C_VEL
LIN {X 0,Y 512.071,Z 395.689,A -85,B 0,C 180,E1 -5467.895,E2 -5467.895} C_VEL
LIN {X 0,Y 515.227,Z 414.042,A -85,B 0,C 180,E1 -5468.312,E2 -5468.312} C_VEL
LIN {X 0,Y 514.005,Z 563.166,A -85,B 0,C 180,E1 -5470.48,E2 -5470.48} C_VEL
LIN {X 0,Y 513.679,Z 578.817,A -85,B 0,C 180,E1 -5470.869,E2 -5470.869} C_VEL
LIN {X 0,Y 513.204,Z 593.479,A -85,B 0,C 180,E1 -5471.389,E2 -5471.389} C_VEL
LIN {X 0,Y 512.71,Z 607.32,A -85,B 0,C 180,E1 -5472.036,E2 -5472.036} C_VEL
LIN {X 0,Y 512.168,Z 621.057,A -85,B 0,C 180,E1 -5472.841,E2 -5472.841} C_VEL
LIN {X 0,Y 511.584,Z 635.016,A -85,B 0,C 180,E1 -5473.848,E2 -5473.848} C_VEL
LIN {X 0,Y 511.07,Z 647.647,A -85,B 0,C 180,E1 -5474.956,E2 -5474.956} C_VEL
LIN {X 0,Y 510.601,Z 658.234,A -85,B 0,C 180,E1 -5476.062,E2 -5476.062} C_VEL
LIN {X 0,Y 510.203,Z 668.062,A -85,B 0,C 180,E1 -5477.267,E2 -5477.267} C_VEL
LIN {X 0,Y 509.856,Z 677.872,A -85,B 0,C 180,E1 -5478.697,E2 -5478.697} C_VEL
LIN {X 0,Y 509.565,Z 685.756,A -85,B 0,C 180,E1 -5480.072,E2 -5480.072} C_VEL
LIN {X 0,Y 509.412,Z 693.266,A -85,B 0,C 180,E1 -5481.67,E2 -5481.67} C_VEL
LIN {X 0,Y 509.29,Z 699.223,A -85,B 0,C 180,E1 -5483.264,E2 -5483.264} C_VEL
LIN {X 0,Y 509.263,Z 702.76,A -85,B 0,C 180,E1 -5484.456,E2 -5484.456} C_VEL
LIN {X 0,Y 509.205,Z 706.339,A -85,B 0,C 180,E1 -5486.043,E2 -5486.043} C_VEL
LIN {X 0,Y 509.186,Z 708.694,A -85,B 0,C 180,E1 -5487.627,E2 -5487.627} C_VEL
LIN {X 0,Y 509.069,Z 709.874,A -85,B 0,C 180,E1 -5489.209,E2 -5489.209} C_VEL
LIN {X 0,Y 509.069,Z 709.876,A -85,B 0,C 180,E1 -5490.791,E2 -5490.791} C_VEL
LIN {X 0,Y 509.186,Z 708.699,A -85,B 0,C 180,E1 -5492.373,E2 -5492.373} C_VEL
LIN {X 0,Y 509.204,Z 706.353,A -85,B 0,C 180,E1 -5493.957,E2 -5493.957} C_VEL
LIN {X 0,Y 509.261,Z 702.792,A -85,B 0,C 180,E1 -5495.543,E2 -5495.543} C_VEL
LIN {X 0,Y 509.314,Z 697.923,A -85,B 0,C 180,E1 -5497.134,E2 -5497.134} C_VEL
LIN {X 0,Y 509.461,Z 691.62,A -85,B 0,C 180,E1 -5498.728,E2 -5498.728} C_VEL
LIN {X 0,Y 509.682,Z 683.705,A -85,B 0,C 180,E1 -5500.326,E2 -5500.326} C_VEL
LIN {X 0,Y 509.932,Z 675.154,A -85,B 0,C 180,E1 -5501.748,E2 -5501.748} C_VEL
LIN {X 0,Y 510.366,Z 665.15,A -85,B 0,C 180,E1 -5503.133,E2 -5503.133} C_VEL
LIN {X 0,Y 510.728,Z 654.79,A -85,B 0,C 180,E1 -5504.341,E2 -5504.341} C_VEL
LIN {X 0,Y 511.263,Z 643.277,A -85,B 0,C 180,E1 -5505.47,E2 -5505.47} C_VEL
LIN {X 0,Y 511.795,Z 630.052,A -85,B 0,C 180,E1 -5506.555,E2 -5506.555} C_VEL
LIN {X 0,Y 512.399,Z 616.566,A -85,B 0,C 180,E1 -5507.459,E2 -5507.459} C_VEL
LIN {X 0,Y 512.974,Z 601.67,A -85,B 0,C 180,E1 -5508.264,E2 -5508.264} C_VEL
LIN {X 0,Y 513.505,Z 586.32,A -85,B 0,C 180,E1 -5508.899,E2 -5508.899} C_VEL
LIN {X 0,Y 513.856,Z 571.448,A -85,B 0,C 180,E1 -5509.349,E2 -5509.349} C_VEL
LIN {X 0,Y 514.1,Z 555.846,A -85,B 0,C 180,E1 -5509.655,E2 -5509.655} C_VEL
LIN {X 0,Y 515.232,Z 418.001,A -85,B 0,C 180,E1 -5511.636,E2 -5511.636} C_VEL
LIN {X 0,Y 515.138,Z 412.752,A -85,B 0,C 180,E1 -5511.719,E2 -5511.719} C_VEL
LIN {X 0,Y 512.128,Z 396.126,A -85,B 0,C 180,E1 -5512.123,E2 -5512.123} C_VEL
LIN {X 0,Y 512.808,Z 375.451,A -85,B 0,C 180,E1 -5514.708,E2 -5514.708} C_VEL
LIN {X 0,Y 513.642,Z 354.324,A -85,B 0,C 180,E1 -5517.386,E2 -5517.386} C_VEL
LIN {X 0,Y 513.186,Z 350.189,A -85,B 0,C 180,E1 -5517.949,E2 -5517.949} C_VEL
LIN {X 0,Y 509.853,Z 336.602,A -85,B 0,C 180,E1 -5519.947,E2 -5519.947} C_VEL
LIN {X 0,Y 509.871,Z 336.597,A -85,B 0,C 180,E1 -5522.774,E2 -5522.774} C_VEL
LIN {X 0,Y 509.823,Z 336.606,A -85,B 0,C 180,E1 -5525.578,E2 -5525.578} C_VEL
LIN {X 0,Y 509.848,Z 336.6,A -85,B 0,C 180,E1 -5528.338,E2 -5528.338} C_VEL
LIN {X 0,Y 509.856,Z 336.601,A -85,B 0,C 180,E1 -5531.425,E2 -5531.425} C_VEL
LIN {X 0,Y 509.854,Z 336.597,A -85,B 0,C 180,E1 -5534.668,E2 -5534.668} C_VEL
LIN {X 0,Y 509.858,Z 336.595,A -85,B 0,C 180,E1 -5538.103,E2 -5538.103} C_VEL
LIN {X 0,Y 509.844,Z 336.598,A -85,B 0,C 180,E1 -5540.648,E2 -5540.648} C_VEL
LIN {X 0,Y 509.833,Z 336.6,A -85,B 0,C 180,E1 -5543.648,E2 -5543.648} C_VEL
LIN {X 0,Y 509.858,Z 336.596,A -85,B 0,C 180,E1 -5546.539,E2 -5546.539} C_VEL
LIN {X 0,Y 509.842,Z 336.602,A -85,B 0,C 180,E1 -5549.334,E2 -5549.334} C_VEL
LIN {X 0,Y 509.889,Z 336.591,A -85,B 0,C 180,E1 -5552.054,E2 -5552.054} C_VEL
LIN {X 0,Y 509.874,Z 336.596,A -85,B 0,C 180,E1 -5554.704,E2 -5554.704} C_VEL
LIN {X 0,Y 509.853,Z 336.599,A -85,B 0,C 180,E1 -5557.45,E2 -5557.45} C_VEL
LIN {X 0,Y 509.914,Z 336.588,A -85,B 0,C 180,E1 -5559.845,E2 -5559.845} C_VEL
LIN {X 0,Y 509.882,Z 336.599,A -85,B 0,C 180,E1 -5563.175,E2 -5563.175} C_VEL
LIN {X 0,Y 509.861,Z 336.595,A -85,B 0,C 180,E1 -5565.634,E2 -5565.634} C_VEL
LIN {X 0,Y 509.899,Z 336.59,A -85,B 0,C 180,E1 -5568.123,E2 -5568.123} C_VEL
LIN {X 0,Y 509.912,Z 336.592,A -85,B 0,C 180,E1 -5571.28,E2 -5571.28} C_VEL
LIN {X 0,Y 509.951,Z 336.584,A -85,B 0,C 180,E1 -5573.67,E2 -5573.67} C_VEL
LIN {X 0,Y 509.953,Z 336.591,A -85,B 0,C 180,E1 -5576.84,E2 -5576.84} C_VEL
LIN {X 0,Y 510.061,Z 336.574,A -85,B 0,C 180,E1 -5579.211,E2 -5579.211} C_VEL
LIN {X 0,Y 510.054,Z 336.572,A -85,B 0,C 180,E1 -5582.369,E2 -5582.369} C_VEL
LIN {X 0,Y 509.98,Z 336.581,A -85,B 0,C 180,E1 -5586.33,E2 -5586.33} C_VEL
LIN {X 0,Y 509.914,Z 336.595,A -85,B 0,C 180,E1 -5588.721,E2 -5588.721} C_VEL
LIN {X 0,Y 509.902,Z 336.589,A -85,B 0,C 180,E1 -5591.932,E2 -5591.932} C_VEL
LIN {X 0,Y 509.892,Z 336.593,A -85,B 0,C 180,E1 -5595.242,E2 -5595.242} C_VEL
LIN {X 0,Y 509.88,Z 336.592,A -85,B 0,C 180,E1 -5597.999,E2 -5597.999} C_VEL
LIN {X 0,Y 509.849,Z 336.601,A -85,B 0,C 180,E1 -5601.002,E2 -5601.002} C_VEL
LIN {X 0,Y 509.86,Z 336.599,A -85,B 0,C 180,E1 -5604.427,E2 -5604.427} C_VEL
LIN {X 0,Y 509.866,Z 336.598,A -85,B 0,C 180,E1 -5607.057,E2 -5607.057} C_VEL
LIN {X 0,Y 509.856,Z 336.595,A -85,B 0,C 180,E1 -5609.752,E2 -5609.752} C_VEL
LIN {X 0,Y 509.872,Z 336.6,A -85,B 0,C 180,E1 -5612.775,E2 -5612.775} C_VEL
LIN {X 0,Y 509.839,Z 336.597,A -85,B 0,C 180,E1 -5615.581,E2 -5615.581} C_VEL
LIN {X 0,Y 509.849,Z 336.6,A -85,B 0,C 180,E1 -5618.339,E2 -5618.339} C_VEL
LIN {X 0,Y 509.852,Z 336.596,A -85,B 0,C 180,E1 -5621.426,E2 -5621.426} C_VEL
LIN {X 0,Y 509.839,Z 336.605,A -85,B 0,C 180,E1 -5624.671,E2 -5624.671} C_VEL
LIN {X 0,Y 509.85,Z 336.598,A -85,B 0,C 180,E1 -5628.105,E2 -5628.105} C_VEL
LIN {X 0,Y 509.846,Z 336.604,A -85,B 0,C 180,E1 -5630.648,E2 -5630.648} C_VEL
LIN {X 0,Y 509.807,Z 336.601,A -85,B 0,C 180,E1 -5633.737,E2 -5633.737} C_VEL
LIN {X 0,Y 509.148,Z 336.69,A -85,B 0,C 180,E1 -5634.397,E2 -5634.397} C_VEL
LIN {X 0,Y 506.342,Z 337.038,A -85,B 0,C 180,E1 -5635.47,E2 -5635.47} C_VEL
LIN {X 0,Y 503.955,Z 337.336,A -85,B 0,C 180,E1 -5636.333,E2 -5636.333} C_VEL
LIN {X 0,Y 502.908,Z 337.463,A -85,B 0,C 180,E1 -5637,E2 -5637} C_VEL
LIN {X 0,Y 502.81,Z 337.473,A -85,B 0,C 180,E1 -5637.225,E2 -5637.225} C_VEL
LIN {X 0,Y 502.816,Z 337.475,A -85,B 0,C 180,E1 -5640.066,E2 -5640.066} C_VEL
LIN {X 0,Y 502.824,Z 337.471,A -85,B 0,C 180,E1 -5643.449,E2 -5643.449} C_VEL
LIN {X 0,Y 502.77,Z 337.482,A -85,B 0,C 180,E1 -5646.086,E2 -5646.086} C_VEL
LIN {X 0,Y 502.784,Z 337.481,A -85,B 0,C 180,E1 -5648.689,E2 -5648.689} C_VEL
LIN {X 0,Y 502.814,Z 337.472,A -85,B 0,C 180,E1 -5651.248,E2 -5651.248} C_VEL
LIN {X 0,Y 502.839,Z 337.474,A -85,B 0,C 180,E1 -5654.665,E2 -5654.665} C_VEL
LIN {X 0,Y 502.881,Z 337.468,A -85,B 0,C 180,E1 -5658.04,E2 -5658.04} C_VEL
LIN {X 0,Y 502.853,Z 337.468,A -85,B 0,C 180,E1 -5661.157,E2 -5661.157} C_VEL
LIN {X 0,Y 502.87,Z 337.466,A -85,B 0,C 180,E1 -5663.581,E2 -5663.581} C_VEL
LIN {X 0,Y 502.838,Z 337.471,A -85,B 0,C 180,E1 -5666.795,E2 -5666.795} C_VEL
LIN {X 0,Y 502.898,Z 337.469,A -85,B 0,C 180,E1 -5668.399,E2 -5668.399} C_VEL
LIN {X 0,Y 502.917,Z 337.461,A -85,B 0,C 180,E1 -5670.801,E2 -5670.801} C_VEL
LIN {X 0,Y 503.012,Z 337.454,A -85,B 0,C 180,E1 -5672.403,E2 -5672.403} C_VEL
LIN {X 0,Y 502.898,Z 337.463,A -85,B 0,C 180,E1 -5675.614,E2 -5675.614} C_VEL
LIN {X 0,Y 502.851,Z 337.474,A -85,B 0,C 180,E1 -5678.034,E2 -5678.034} C_VEL
LIN {X 0,Y 502.84,Z 337.47,A -85,B 0,C 180,E1 -5681.284,E2 -5681.284} C_VEL
LIN {X 0,Y 502.801,Z 337.48,A -85,B 0,C 180,E1 -5684.572,E2 -5684.572} C_VEL
LIN {X 0,Y 502.76,Z 337.51,A -85,B 0,C 180,E1 -5686.548,E2 -5686.548} C_VEL
LIN {X 0,Y 504.034,Z 343.249,A -85,B 0,C 180,E1 -5687.602,E2 -5687.602} C_VEL
LIN {X 0,Y 507.562,Z 352.976,A -85,B 0,C 180,E1 -5687.918,E2 -5687.918} C_VEL
LIN {X 0,Y 508.762,Z 358.372,A -85,B 0,C 180,E1 -5688.057,E2 -5688.057} C_VEL
LIN {X 0,Y 507.463,Z 507.738,A -85,B 0,C 180,E1 -5690.271,E2 -5690.271} C_VEL
LIN {X 0,Y 507.148,Z 523.339,A -85,B 0,C 180,E1 -5690.668,E2 -5690.668} C_VEL
LIN {X 0,Y 506.77,Z 537.727,A -85,B 0,C 180,E1 -5691.195,E2 -5691.195} C_VEL
LIN {X 0,Y 506.261,Z 551.979,A -85,B 0,C 180,E1 -5691.882,E2 -5691.882} C_VEL
LIN {X 0,Y 505.686,Z 565.239,A -85,B 0,C 180,E1 -5692.686,E2 -5692.686} C_VEL
LIN {X 0,Y 505.139,Z 576.623,A -85,B 0,C 180,E1 -5693.521,E2 -5693.521} C_VEL
LIN {X 0,Y 504.563,Z 588.822,A -85,B 0,C 180,E1 -5694.591,E2 -5694.591} C_VEL
LIN {X 0,Y 503.975,Z 600.638,A -85,B 0,C 180,E1 -5695.836,E2 -5695.836} C_VEL
LIN {X 0,Y 503.432,Z 611.666,A -85,B 0,C 180,E1 -5697.236,E2 -5697.236} C_VEL
LIN {X 0,Y 503.031,Z 620.535,A -85,B 0,C 180,E1 -5698.589,E2 -5698.589} C_VEL
LIN {X 0,Y 502.655,Z 629.373,A -85,B 0,C 180,E1 -5700.222,E2 -5700.222} C_VEL
LIN {X 0,Y 502.442,Z 636.029,A -85,B 0,C 180,E1 -5701.739,E2 -5701.739} C_VEL
LIN {X 0,Y 502.261,Z 640.826,A -85,B 0,C 180,E1 -5703.074,E2 -5703.074} C_VEL
LIN {X 0,Y 502.177,Z 644.455,A -85,B 0,C 180,E1 -5704.339,E2 -5704.339} C_VEL
LIN {X 0,Y 502.015,Z 648.104,A -85,B 0,C 180,E1 -5706.014,E2 -5706.014} C_VEL
LIN {X 0,Y 501.99,Z 649.721,A -85,B 0,C 180,E1 -5707.058,E2 -5707.058} C_VEL
LIN {X 0,Y 501.989,Z 651.08,A -85,B 0,C 180,E1 -5708.369,E2 -5708.369} C_VEL
LIN {X 0,Y 501.976,Z 651.711,A -85,B 0,C 180,E1 -5710.093,E2 -5710.093} C_VEL
LIN {X 0,Y 501.985,Z 651.43,A -85,B 0,C 180,E1 -5711.149,E2 -5711.149} C_VEL
LIN {X 0,Y 501.99,Z 650.658,A -85,B 0,C 180,E1 -5712.223,E2 -5712.223} C_VEL
LIN {X 0,Y 502.061,Z 649.375,A -85,B 0,C 180,E1 -5713.308,E2 -5713.308} C_VEL
LIN {X 0,Y 502.169,Z 646.364,A -85,B 0,C 180,E1 -5714.972,E2 -5714.972} C_VEL
LIN {X 0,Y 502.279,Z 641.808,A -85,B 0,C 180,E1 -5716.715,E2 -5716.715} C_VEL
LIN {X 0,Y 502.428,Z 635.994,A -85,B 0,C 180,E1 -5718.384,E2 -5718.384} C_VEL
LIN {X 0,Y 502.683,Z 628.978,A -85,B 0,C 180,E1 -5719.974,E2 -5719.974} C_VEL
LIN {X 0,Y 503.046,Z 620.814,A -85,B 0,C 180,E1 -5721.478,E2 -5721.478} C_VEL
LIN {X 0,Y 503.486,Z 611.343,A -85,B 0,C 180,E1 -5722.921,E2 -5722.921} C_VEL
LIN {X 0,Y 503.999,Z 600.669,A -85,B 0,C 180,E1 -5724.272,E2 -5724.272} C_VEL
LIN {X 0,Y 504.584,Z 589.302,A -85,B 0,C 180,E1 -5725.472,E2 -5725.472} C_VEL
LIN {X 0,Y 505.158,Z 576.578,A -85,B 0,C 180,E1 -5726.59,E2 -5726.59} C_VEL
LIN {X 0,Y 505.797,Z 562.727,A -85,B 0,C 180,E1 -5727.584,E2 -5727.584} C_VEL
LIN {X 0,Y 506.384,Z 548.457,A -85,B 0,C 180,E1 -5728.404,E2 -5728.404} C_VEL
LIN {X 0,Y 506.826,Z 534.931,A -85,B 0,C 180,E1 -5729.015,E2 -5729.015} C_VEL
LIN {X 0,Y 507.198,Z 519.732,A -85,B 0,C 180,E1 -5729.531,E2 -5729.531} C_VEL
LIN {X 0,Y 507.503,Z 504.232,A -85,B 0,C 180,E1 -5729.882,E2 -5729.882} C_VEL
LIN {X 0,Y 508.8,Z 358.125,A -85,B 0,C 180,E1 -5732.045,E2 -5732.045} C_VEL
LIN {X 0,Y 506.753,Z 350.491,A -85,B 0,C 180,E1 -5732.259,E2 -5732.259} C_VEL
LIN {X 0,Y 504.195,Z 343.937,A -85,B 0,C 180,E1 -5732.501,E2 -5732.501} C_VEL
LIN {X 0,Y 502.777,Z 337.484,A -85,B 0,C 180,E1 -5733.736,E2 -5733.736} C_VEL
LIN {X 0,Y 502.785,Z 337.48,A -85,B 0,C 180,E1 -5736.959,E2 -5736.959} C_VEL
LIN {X 0,Y 502.831,Z 337.476,A -85,B 0,C 180,E1 -5739.548,E2 -5739.548} C_VEL
LIN {X 0,Y 502.803,Z 337.478,A -85,B 0,C 180,E1 -5742.091,E2 -5742.091} C_VEL
LIN {X 0,Y 502.834,Z 337.476,A -85,B 0,C 180,E1 -5745.429,E2 -5745.429} C_VEL
LIN {X 0,Y 502.878,Z 337.466,A -85,B 0,C 180,E1 -5748.717,E2 -5748.717} C_VEL
LIN {X 0,Y 502.852,Z 337.473,A -85,B 0,C 180,E1 -5751.966,E2 -5751.966} C_VEL
LIN {X 0,Y 502.9,Z 337.463,A -85,B 0,C 180,E1 -5754.386,E2 -5754.386} C_VEL
LIN {X 0,Y 503.014,Z 337.455,A -85,B 0,C 180,E1 -5757.597,E2 -5757.597} C_VEL
LIN {X 0,Y 502.972,Z 337.455,A -85,B 0,C 180,E1 -5760.8,E2 -5760.8} C_VEL
LIN {X 0,Y 503.021,Z 337.447,A -85,B 0,C 180,E1 -5762.402,E2 -5762.402} C_VEL
LIN {X 0,Y 502.92,Z 337.467,A -85,B 0,C 180,E1 -5765.613,E2 -5765.613} C_VEL
LIN {X 0,Y 502.865,Z 337.469,A -85,B 0,C 180,E1 -5768.843,E2 -5768.843} C_VEL
LIN {X 0,Y 502.848,Z 337.469,A -85,B 0,C 180,E1 -5772.101,E2 -5772.101} C_VEL
LIN {X 0,Y 502.851,Z 337.473,A -85,B 0,C 180,E1 -5775.399,E2 -5775.399} C_VEL
LIN {X 0,Y 502.829,Z 337.472,A -85,B 0,C 180,E1 -5778.752,E2 -5778.752} C_VEL
LIN {X 0,Y 502.785,Z 337.482,A -85,B 0,C 180,E1 -5781.311,E2 -5781.311} C_VEL
LIN {X 0,Y 502.779,Z 337.477,A -85,B 0,C 180,E1 -5783.914,E2 -5783.914} C_VEL
LIN {X 0,Y 502.866,Z 337.468,A -85,B 0,C 180,E1 -5786.566,E2 -5786.566} C_VEL
LIN {X 0,Y 502.826,Z 337.476,A -85,B 0,C 180,E1 -5789.287,E2 -5789.287} C_VEL
LIN {X 0,Y 502.785,Z 337.476,A -85,B 0,C 180,E1 -5792.084,E2 -5792.084} C_VEL
LIN {X 0,Y 502.8,Z 337.481,A -85,B 0,C 180,E1 -5794.965,E2 -5794.965} C_VEL
LIN {X 0,Y 502.795,Z 337.477,A -85,B 0,C 180,E1 -5797.954,E2 -5797.954} C_VEL
LIN {X 0,Y 502.822,Z 337.479,A -85,B 0,C 180,E1 -5801.065,E2 -5801.065} C_VEL
LIN {X 0,Y 502.802,Z 337.479,A -85,B 0,C 180,E1 -5804.531,E2 -5804.531} C_VEL
LIN {X 0,Y 502.832,Z 337.472,A -85,B 0,C 180,E1 -5807.864,E2 -5807.864} C_VEL
LIN {X 0,Y 502.803,Z 337.48,A -85,B 0,C 180,E1 -5811.024,E2 -5811.024} C_VEL
LIN {X 0,Y 502.776,Z 337.481,A -85,B 0,C 180,E1 -5814.169,E2 -5814.169} C_VEL
LIN {X 0,Y 502.834,Z 337.478,A -85,B 0,C 180,E1 -5816.993,E2 -5816.993} C_VEL
LIN {X 0,Y 502.851,Z 337.62,A -85,B 0,C 180,E1 -5819.921,E2 -5819.921} C_VEL
LIN {X 0,Y 506.363,Z 352.158,A -85,B 0,C 180,E1 -5822.066,E2 -5822.066} C_VEL
LIN {X 0,Y 506.608,Z 356.142,A -85,B 0,C 180,E1 -5822.604,E2 -5822.604} C_VEL
LIN {X 0,Y 505.78,Z 377.671,A -85,B 0,C 180,E1 -5825.363,E2 -5825.363} C_VEL
LIN {X 0,Y 505.168,Z 395.176,A -85,B 0,C 180,E1 -5827.572,E2 -5827.572} C_VEL
LIN {X 0,Y 508.616,Z 415.521,A -85,B 0,C 180,E1 -5828.046,E2 -5828.046} C_VEL
LIN {X 0,Y 507.295,Z 563.079,A -85,B 0,C 180,E1 -5830.226,E2 -5830.226} C_VEL
LIN {X 0,Y 506.92,Z 578.724,A -85,B 0,C 180,E1 -5830.623,E2 -5830.623} C_VEL
LIN {X 0,Y 506.434,Z 593.265,A -85,B 0,C 180,E1 -5831.148,E2 -5831.148} C_VEL
LIN {X 0,Y 505.923,Z 606.731,A -85,B 0,C 180,E1 -5831.786,E2 -5831.786} C_VEL
LIN {X 0,Y 505.322,Z 620.498,A -85,B 0,C 180,E1 -5832.601,E2 -5832.601} C_VEL
LIN {X 0,Y 504.688,Z 634.481,A -85,B 0,C 180,E1 -5833.621,E2 -5833.621} C_VEL
LIN {X 0,Y 504.087,Z 647.129,A -85,B 0,C 180,E1 -5834.742,E2 -5834.742} C_VEL
LIN {X 0,Y 503.605,Z 657.735,A -85,B 0,C 180,E1 -5835.864,E2 -5835.864} C_VEL
LIN {X 0,Y 503.194,Z 667.578,A -85,B 0,C 180,E1 -5837.087,E2 -5837.087} C_VEL
LIN {X 0,Y 502.806,Z 677.483,A -85,B 0,C 180,E1 -5838.55,E2 -5838.55} C_VEL
LIN {X 0,Y 502.521,Z 685.299,A -85,B 0,C 180,E1 -5839.932,E2 -5839.932} C_VEL
LIN {X 0,Y 502.338,Z 692.82,A -85,B 0,C 180,E1 -5841.552,E2 -5841.552} C_VEL
LIN {X 0,Y 502.223,Z 698.788,A -85,B 0,C 180,E1 -5843.169,E2 -5843.169} C_VEL
LIN {X 0,Y 502.176,Z 702.331,A -85,B 0,C 180,E1 -5844.378,E2 -5844.378} C_VEL
LIN {X 0,Y 502.104,Z 705.916,A -85,B 0,C 180,E1 -5845.986,E2 -5845.986} C_VEL
LIN {X 0,Y 502.117,Z 708.279,A -85,B 0,C 180,E1 -5847.593,E2 -5847.593} C_VEL
LIN {X 0,Y 501.987,Z 709.464,A -85,B 0,C 180,E1 -5849.197,E2 -5849.197} C_VEL
LIN {X 0,Y 501.987,Z 709.469,A -85,B 0,C 180,E1 -5850.802,E2 -5850.802} C_VEL
LIN {X 0,Y 502.117,Z 708.293,A -85,B 0,C 180,E1 -5852.406,E2 -5852.406} C_VEL
LIN {X 0,Y 502.103,Z 705.945,A -85,B 0,C 180,E1 -5854.013,E2 -5854.013} C_VEL
LIN {X 0,Y 502.171,Z 702.383,A -85,B 0,C 180,E1 -5855.622,E2 -5855.622} C_VEL
LIN {X 0,Y 502.24,Z 697.511,A -85,B 0,C 180,E1 -5857.235,E2 -5857.235} C_VEL
LIN {X 0,Y 502.37,Z 691.201,A -85,B 0,C 180,E1 -5858.852,E2 -5858.852} C_VEL
LIN {X 0,Y 502.641,Z 683.281,A -85,B 0,C 180,E1 -5860.472,E2 -5860.472} C_VEL
LIN {X 0,Y 502.897,Z 674.34,A -85,B 0,C 180,E1 -5861.972,E2 -5861.972} C_VEL
LIN {X 0,Y 503.354,Z 664.709,A -85,B 0,C 180,E1 -5863.319,E2 -5863.319} C_VEL
LIN {X 0,Y 503.757,Z 654.344,A -85,B 0,C 180,E1 -5864.543,E2 -5864.543} C_VEL
LIN {X 0,Y 504.355,Z 642.227,A -85,B 0,C 180,E1 -5865.744,E2 -5865.744} C_VEL
LIN {X 0,Y 504.914,Z 629.583,A -85,B 0,C 180,E1 -5866.787,E2 -5866.787} C_VEL
LIN {X 0,Y 505.574,Z 616.082,A -85,B 0,C 180,E1 -5867.703,E2 -5867.703} C_VEL
LIN {X 0,Y 506.175,Z 601.159,A -85,B 0,C 180,E1 -5868.518,E2 -5868.518} C_VEL
LIN {X 0,Y 506.769,Z 585.579,A -85,B 0,C 180,E1 -5869.167,E2 -5869.167} C_VEL
LIN {X 0,Y 507.144,Z 570.84,A -85,B 0,C 180,E1 -5869.615,E2 -5869.615} C_VEL
LIN {X 0,Y 507.381,Z 555.962,A -85,B 0,C 180,E1 -5869.911,E2 -5869.911} C_VEL
LIN {X 0,Y 508.647,Z 415.057,A -85,B 0,C 180,E1 -5871.97,E2 -5871.97} C_VEL
LIN {X 0,Y 505.274,Z 395.744,A -85,B 0,C 180,E1 -5872.44,E2 -5872.44} C_VEL
LIN {X 0,Y 506.247,Z 371.387,A -85,B 0,C 180,E1 -5875.529,E2 -5875.529} C_VEL
LIN {X 0,Y 506.837,Z 354.509,A -85,B 0,C 180,E1 -5877.712,E2 -5877.712} C_VEL
LIN {X 0,Y 503.767,Z 341.389,A -85,B 0,C 180,E1 -5879.636,E2 -5879.636} C_VEL
LIN {X 0,Y 502.821,Z 337.478,A -85,B 0,C 180,E1 -5880.239,E2 -5880.239} C_VEL
LIN {X 0,Y 502.829,Z 337.477,A -85,B 0,C 180,E1 -5883.031,E2 -5883.031} C_VEL
LIN {X 0,Y 502.771,Z 337.482,A -85,B 0,C 180,E1 -5885.951,E2 -5885.951} C_VEL
LIN {X 0,Y 502.8,Z 337.483,A -85,B 0,C 180,E1 -5888.976,E2 -5888.976} C_VEL
LIN {X 0,Y 502.827,Z 337.471,A -85,B 0,C 180,E1 -5892.136,E2 -5892.136} C_VEL
LIN {X 0,Y 502.798,Z 337.479,A -85,B 0,C 180,E1 -5895.468,E2 -5895.468} C_VEL
LIN {X 0,Y 502.827,Z 337.472,A -85,B 0,C 180,E1 -5897.864,E2 -5897.864} C_VEL
LIN {X 0,Y 502.799,Z 337.481,A -85,B 0,C 180,E1 -5901.024,E2 -5901.024} C_VEL
LIN {X 0,Y 502.783,Z 337.476,A -85,B 0,C 180,E1 -5904.167,E2 -5904.167} C_VEL
LIN {X 0,Y 502.829,Z 337.477,A -85,B 0,C 180,E1 -5906.993,E2 -5906.993} C_VEL
LIN {X 0,Y 502.811,Z 337.472,A -85,B 0,C 180,E1 -5910.065,E2 -5910.065} C_VEL
LIN {X 0,Y 502.829,Z 337.472,A -85,B 0,C 180,E1 -5912.533,E2 -5912.533} C_VEL
LIN {X 0,Y 502.826,Z 337.476,A -85,B 0,C 180,E1 -5915.298,E2 -5915.298} C_VEL
LIN {X 0,Y 502.791,Z 337.475,A -85,B 0,C 180,E1 -5917.827,E2 -5917.827} C_VEL
LIN {X 0,Y 502.822,Z 337.472,A -85,B 0,C 180,E1 -5920.4,E2 -5920.4} C_VEL
LIN {X 0,Y 502.831,Z 337.478,A -85,B 0,C 180,E1 -5922.932,E2 -5922.932} C_VEL
LIN {X 0,Y 502.842,Z 337.472,A -85,B 0,C 180,E1 -5925.429,E2 -5925.429} C_VEL
LIN {X 0,Y 502.875,Z 337.47,A -85,B 0,C 180,E1 -5928.717,E2 -5928.717} C_VEL
LIN {X 0,Y 502.899,Z 337.461,A -85,B 0,C 180,E1 -5931.967,E2 -5931.967} C_VEL
LIN {X 0,Y 502.931,Z 337.459,A -85,B 0,C 180,E1 -5934.387,E2 -5934.387} C_VEL
LIN {X 0,Y 503.023,Z 337.447,A -85,B 0,C 180,E1 -5937.598,E2 -5937.598} C_VEL
LIN {X 0,Y 503.025,Z 337.446,A -85,B 0,C 180,E1 -5940,E2 -5940} C_VEL
LIN {X 0,Y 503.023,Z 337.448,A -85,B 0,C 180,E1 -5942.403,E2 -5942.403} C_VEL
LIN {X 0,Y 502.938,Z 337.457,A -85,B 0,C 180,E1 -5945.614,E2 -5945.614} C_VEL
LIN {X 0,Y 502.9,Z 337.462,A -85,B 0,C 180,E1 -5948.034,E2 -5948.034} C_VEL
LIN {X 0,Y 502.875,Z 337.467,A -85,B 0,C 180,E1 -5951.284,E2 -5951.284} C_VEL
LIN {X 0,Y 502.843,Z 337.474,A -85,B 0,C 180,E1 -5954.571,E2 -5954.571} C_VEL
LIN {X 0,Y 502.854,Z 337.467,A -85,B 0,C 180,E1 -5957.908,E2 -5957.908} C_VEL
LIN {X 0,Y 502.827,Z 337.476,A -85,B 0,C 180,E1 -5960.537,E2 -5960.537} C_VEL
LIN {X 0,Y 502.789,Z 337.48,A -85,B 0,C 180,E1 -5963.041,E2 -5963.041} C_VEL
LIN {X 0,Y 502.809,Z 337.473,A -85,B 0,C 180,E1 -5965.678,E2 -5965.678} C_VEL
LIN {X 0,Y 502.834,Z 337.474,A -85,B 0,C 180,E1 -5968.373,E2 -5968.373} C_VEL
LIN {X 0,Y 502.792,Z 337.475,A -85,B 0,C 180,E1 -5971.499,E2 -5971.499} C_VEL
LIN {X 0,Y 502.804,Z 337.479,A -85,B 0,C 180,E1 -5974.445,E2 -5974.445} C_VEL
LIN {X 0,Y 502.78,Z 337.478,A -85,B 0,C 180,E1 -5977.179,E2 -5977.179} C_VEL
LIN {X 0,Y 502.787,Z 337.477,A -85,B 0,C 180,E1 -5980.016,E2 -5980.016} C_VEL
LIN {X 0,Y 502.803,Z 337.477,A -85,B 0,C 180,E1 -5982.2,E2 -5982.2} C_VEL
LIN {X 0,Y 502.786,Z 337.476,A -85,B 0,C 180,E1 -5985.471,E2 -5985.471} C_VEL
LIN {X 0,Y 502.795,Z 337.475,A -85,B 0,C 180,E1 -5987.861,E2 -5987.861} C_VEL
LIN {X 0,Y 502.801,Z 337.476,A -85,B 0,C 180,E1 -5991.024,E2 -5991.024} C_VEL
LIN {X 0,Y 502.772,Z 337.481,A -85,B 0,C 180,E1 -5994.17,E2 -5994.17} C_VEL
LIN {X 0,Y 502.81,Z 337.473,A -85,B 0,C 180,E1 -5997.225,E2 -5997.225} C_VEL
LIN {X 0,Y 502.109,Z 337.563,A -85,B 0,C 180,E1 -5997.894,E2 -5997.894} C_VEL
LIN {X 0,Y 499.247,Z 337.919,A -85,B 0,C 180,E1 -5998.98,E2 -5998.98} C_VEL
LIN {X 0,Y 496.848,Z 338.218,A -85,B 0,C 180,E1 -5999.855,E2 -5999.855} C_VEL
LIN {X 0,Y 495.821,Z 338.351,A -85,B 0,C 180,E1 -6000.53,E2 -6000.53} C_VEL
LIN {X 0,Y 495.738,Z 338.355,A -85,B 0,C 180,E1 -6000.759,E2 -6000.759} C_VEL
LIN {X 0,Y 495.745,Z 338.355,A -85,B 0,C 180,E1 -6003.93,E2 -6003.93} C_VEL
LIN {X 0,Y 495.761,Z 338.351,A -85,B 0,C 180,E1 -6007.14,E2 -6007.14} C_VEL
LIN {X 0,Y 495.77,Z 338.354,A -85,B 0,C 180,E1 -6010.11,E2 -6010.11} C_VEL
LIN {X 0,Y 495.717,Z 338.361,A -85,B 0,C 180,E1 -6012.679,E2 -6012.679} C_VEL
LIN {X 0,Y 495.783,Z 338.348,A -85,B 0,C 180,E1 -6015.217,E2 -6015.217} C_VEL
LIN {X 0,Y 495.854,Z 338.345,A -85,B 0,C 180,E1 -6018.555,E2 -6018.555} C_VEL
LIN {X 0,Y 495.817,Z 338.346,A -85,B 0,C 180,E1 -6021.852,E2 -6021.852} C_VEL
LIN {X 0,Y 495.855,Z 338.348,A -85,B 0,C 180,E1 -6024.306,E2 -6024.306} C_VEL
LIN {X 0,Y 495.98,Z 338.324,A -85,B 0,C 180,E1 -6027.564,E2 -6027.564} C_VEL
LIN {X 0,Y 495.976,Z 338.329,A -85,B 0,C 180,E1 -6030,E2 -6030} C_VEL
LIN {X 0,Y 495.979,Z 338.33,A -85,B 0,C 180,E1 -6032.437,E2 -6032.437} C_VEL
LIN {X 0,Y 495.856,Z 338.341,A -85,B 0,C 180,E1 -6035.694,E2 -6035.694} C_VEL
LIN {X 0,Y 495.815,Z 338.352,A -85,B 0,C 180,E1 -6038.149,E2 -6038.149} C_VEL
LIN {X 0,Y 495.825,Z 338.345,A -85,B 0,C 180,E1 -6041.446,E2 -6041.446} C_VEL
LIN {X 0,Y 495.749,Z 338.359,A -85,B 0,C 180,E1 -6044.784,E2 -6044.784} C_VEL
LIN {X 0,Y 495.73,Z 338.524,A -85,B 0,C 180,E1 -6046.313,E2 -6046.313} C_VEL
LIN {X 0,Y 496.863,Z 343.524,A -85,B 0,C 180,E1 -6047.254,E2 -6047.254} C_VEL
LIN {X 0,Y 501.188,Z 354.962,A -85,B 0,C 180,E1 -6047.649,E2 -6047.649} C_VEL
LIN {X 0,Y 502.24,Z 360.31,A -85,B 0,C 180,E1 -6047.781,E2 -6047.781} C_VEL
LIN {X 0,Y 500.77,Z 508.479,A -85,B 0,C 180,E1 -6050.01,E2 -6050.01} C_VEL
LIN {X 0,Y 500.448,Z 523.695,A -85,B 0,C 180,E1 -6050.404,E2 -6050.404} C_VEL
LIN {X 0,Y 500.041,Z 538.336,A -85,B 0,C 180,E1 -6050.948,E2 -6050.948} C_VEL
LIN {X 0,Y 499.509,Z 552.214,A -85,B 0,C 180,E1 -6051.626,E2 -6051.626} C_VEL
LIN {X 0,Y 498.9,Z 565.865,A -85,B 0,C 180,E1 -6052.465,E2 -6052.465} C_VEL
LIN {X 0,Y 498.269,Z 578.32,A -85,B 0,C 180,E1 -6053.401,E2 -6053.401} C_VEL
LIN {X 0,Y 497.622,Z 590.575,A -85,B 0,C 180,E1 -6054.511,E2 -6054.511} C_VEL
LIN {X 0,Y 497.022,Z 602.273,A -85,B 0,C 180,E1 -6055.786,E2 -6055.786} C_VEL
LIN {X 0,Y 496.438,Z 612.813,A -85,B 0,C 180,E1 -6057.166,E2 -6057.166} C_VEL
LIN {X 0,Y 496.035,Z 621.596,A -85,B 0,C 180,E1 -6058.545,E2 -6058.545} C_VEL
LIN {X 0,Y 495.625,Z 629.925,A -85,B 0,C 180,E1 -6060.118,E2 -6060.118} C_VEL
LIN {X 0,Y 495.416,Z 636.561,A -85,B 0,C 180,E1 -6061.661,E2 -6061.661} C_VEL
LIN {X 0,Y 495.183,Z 641.699,A -85,B 0,C 180,E1 -6063.136,E2 -6063.136} C_VEL
LIN {X 0,Y 495.077,Z 645.721,A -85,B 0,C 180,E1 -6064.599,E2 -6064.599} C_VEL
LIN {X 0,Y 494.935,Z 648.513,A -85,B 0,C 180,E1 -6065.963,E2 -6065.963} C_VEL
LIN {X 0,Y 494.895,Z 650.845,A -85,B 0,C 180,E1 -6067.636,E2 -6067.636} C_VEL
LIN {X 0,Y 494.906,Z 651.677,A -85,B 0,C 180,E1 -6068.67,E2 -6068.67} C_VEL
LIN {X 0,Y 494.887,Z 652.107,A -85,B 0,C 180,E1 -6069.926,E2 -6069.926} C_VEL
LIN {X 0,Y 494.911,Z 651.433,A -85,B 0,C 180,E1 -6071.869,E2 -6071.869} C_VEL
LIN {X 0,Y 494.991,Z 649.452,A -85,B 0,C 180,E1 -6073.605,E2 -6073.605} C_VEL
LIN {X 0,Y 495.111,Z 646.406,A -85,B 0,C 180,E1 -6075.214,E2 -6075.214} C_VEL
LIN {X 0,Y 495.212,Z 642.495,A -85,B 0,C 180,E1 -6076.718,E2 -6076.718} C_VEL
LIN {X 0,Y 495.391,Z 636.425,A -85,B 0,C 180,E1 -6078.497,E2 -6078.497} C_VEL
LIN {X 0,Y 495.648,Z 630.09,A -85,B 0,C 180,E1 -6079.969,E2 -6079.969} C_VEL
LIN {X 0,Y 496.01,Z 622.444,A -85,B 0,C 180,E1 -6081.432,E2 -6081.432} C_VEL
LIN {X 0,Y 496.461,Z 614.171,A -85,B 0,C 180,E1 -6082.758,E2 -6082.758} C_VEL
LIN {X 0,Y 496.978,Z 603.473,A -85,B 0,C 180,E1 -6084.189,E2 -6084.189} C_VEL
LIN {X 0,Y 497.627,Z 591.95,A -85,B 0,C 180,E1 -6085.466,E2 -6085.466} C_VEL
LIN {X 0,Y 498.242,Z 579.375,A -85,B 0,C 180,E1 -6086.624,E2 -6086.624} C_VEL
LIN {X 0,Y 498.914,Z 565.985,A -85,B 0,C 180,E1 -6087.636,E2 -6087.636} C_VEL
LIN {X 0,Y 499.535,Z 552.693,A -85,B 0,C 180,E1 -6088.453,E2 -6088.453} C_VEL
LIN {X 0,Y 499.995,Z 538.595,A -85,B 0,C 180,E1 -6089.144,E2 -6089.144} C_VEL
LIN {X 0,Y 500.453,Z 523.426,A -85,B 0,C 180,E1 -6089.702,E2 -6089.702} C_VEL
LIN {X 0,Y 500.788,Z 507.273,A -85,B 0,C 180,E1 -6090.106,E2 -6090.106} C_VEL
LIN {X 0,Y 502.284,Z 359.629,A -85,B 0,C 180,E1 -6092.33,E2 -6092.33} C_VEL
LIN {X 0,Y 500.587,Z 353.23,A -85,B 0,C 180,E1 -6092.512,E2 -6092.512} C_VEL
LIN {X 0,Y 497.089,Z 344.421,A -85,B 0,C 180,E1 -6092.842,E2 -6092.842} C_VEL
LIN {X 0,Y 495.747,Z 338.361,A -85,B 0,C 180,E1 -6094.042,E2 -6094.042} C_VEL
LIN {X 0,Y 495.736,Z 338.36,A -85,B 0,C 180,E1 -6097.494,E2 -6097.494} C_VEL
LIN {X 0,Y 495.757,Z 338.356,A -85,B 0,C 180,E1 -6100.109,E2 -6100.109} C_VEL
LIN {X 0,Y 495.717,Z 338.356,A -85,B 0,C 180,E1 -6102.679,E2 -6102.679} C_VEL
LIN {X 0,Y 495.783,Z 338.352,A -85,B 0,C 180,E1 -6105.217,E2 -6105.217} C_VEL
LIN {X 0,Y 495.853,Z 338.342,A -85,B 0,C 180,E1 -6108.555,E2 -6108.555} C_VEL
LIN {X 0,Y 495.816,Z 338.351,A -85,B 0,C 180,E1 -6111.851,E2 -6111.851} C_VEL
LIN {X 0,Y 495.858,Z 338.341,A -85,B 0,C 180,E1 -6114.306,E2 -6114.306} C_VEL
LIN {X 0,Y 495.981,Z 338.33,A -85,B 0,C 180,E1 -6117.563,E2 -6117.563} C_VEL
LIN {X 0,Y 496,Z 338.325,A -85,B 0,C 180,E1 -6120,E2 -6120} C_VEL
LIN {X 0,Y 495.989,Z 338.323,A -85,B 0,C 180,E1 -6122.436,E2 -6122.436} C_VEL
LIN {X 0,Y 495.875,Z 338.343,A -85,B 0,C 180,E1 -6125.693,E2 -6125.693} C_VEL
LIN {X 0,Y 495.835,Z 338.346,A -85,B 0,C 180,E1 -6128.97,E2 -6128.97} C_VEL
LIN {X 0,Y 495.831,Z 338.343,A -85,B 0,C 180,E1 -6132.034,E2 -6132.034} C_VEL
LIN {X 0,Y 495.826,Z 338.347,A -85,B 0,C 180,E1 -6135.451,E2 -6135.451} C_VEL
LIN {X 0,Y 495.781,Z 338.348,A -85,B 0,C 180,E1 -6138.237,E2 -6138.237} C_VEL
LIN {X 0,Y 495.777,Z 338.352,A -85,B 0,C 180,E1 -6140.756,E2 -6140.756} C_VEL
LIN {X 0,Y 495.745,Z 338.358,A -85,B 0,C 180,E1 -6143.387,E2 -6143.387} C_VEL
LIN {X 0,Y 495.792,Z 338.348,A -85,B 0,C 180,E1 -6146.068,E2 -6146.068} C_VEL
LIN {X 0,Y 495.774,Z 338.355,A -85,B 0,C 180,E1 -6148.814,E2 -6148.814} C_VEL
LIN {X 0,Y 495.757,Z 338.353,A -85,B 0,C 180,E1 -6151.725,E2 -6151.725} C_VEL
LIN {X 0,Y 495.77,Z 338.355,A -85,B 0,C 180,E1 -6154.694,E2 -6154.694} C_VEL
LIN {X 0,Y 495.731,Z 338.359,A -85,B 0,C 180,E1 -6157.561,E2 -6157.561} C_VEL
LIN {X 0,Y 495.768,Z 338.357,A -85,B 0,C 180,E1 -6160.699,E2 -6160.699} C_VEL
LIN {X 0,Y 495.736,Z 338.356,A -85,B 0,C 180,E1 -6164.001,E2 -6164.001} C_VEL
LIN {X 0,Y 495.735,Z 338.361,A -85,B 0,C 180,E1 -6167.117,E2 -6167.117} C_VEL
LIN {X 0,Y 495.76,Z 338.355,A -85,B 0,C 180,E1 -6169.953,E2 -6169.953} C_VEL
LIN {X 0,Y 495.729,Z 338.363,A -85,B 0,C 180,E1 -6172.553,E2 -6172.553} C_VEL
LIN {X 0,Y 495.779,Z 338.354,A -85,B 0,C 180,E1 -6175.456,E2 -6175.456} C_VEL
LIN {X 0,Y 495.756,Z 338.358,A -85,B 0,C 180,E1 -6178.363,E2 -6178.363} C_VEL
LIN {X 0,Y 495.809,Z 338.496,A -85,B 0,C 180,E1 -6179.622,E2 -6179.622} C_VEL
LIN {X 0,Y 499.762,Z 355.181,A -85,B 0,C 180,E1 -6182.122,E2 -6182.122} C_VEL
LIN {X 0,Y 499.291,Z 370.45,A -85,B 0,C 180,E1 -6184.128,E2 -6184.128} C_VEL
LIN {X 0,Y 498.352,Z 394.194,A -85,B 0,C 180,E1 -6187.181,E2 -6187.181} C_VEL
LIN {X 0,Y 498.399,Z 395.276,A -85,B 0,C 180,E1 -6187.264,E2 -6187.264} C_VEL
LIN {X 0,Y 502.009,Z 416.182,A -85,B 0,C 180,E1 -6187.759,E2 -6187.759} C_VEL
LIN {X 0,Y 500.601,Z 561.524,A -85,B 0,C 180,E1 -6189.935,E2 -6189.935} C_VEL
LIN {X 0,Y 500.212,Z 576.919,A -85,B 0,C 180,E1 -6190.317,E2 -6190.317} C_VEL
LIN {X 0,Y 499.676,Z 591.927,A -85,B 0,C 180,E1 -6190.854,E2 -6190.854} C_VEL
LIN {X 0,Y 499.082,Z 606.136,A -85,B 0,C 180,E1 -6191.528,E2 -6191.528} C_VEL
LIN {X 0,Y 498.477,Z 619.939,A -85,B 0,C 180,E1 -6192.354,E2 -6192.354} C_VEL
LIN {X 0,Y 497.823,Z 632.634,A -85,B 0,C 180,E1 -6193.283,E2 -6193.283} C_VEL
LIN {X 0,Y 497.282,Z 644.305,A -85,B 0,C 180,E1 -6194.305,E2 -6194.305} C_VEL
LIN {X 0,Y 496.674,Z 655.421,A -85,B 0,C 180,E1 -6195.453,E2 -6195.453} C_VEL
LIN {X 0,Y 496.237,Z 665.584,A -85,B 0,C 180,E1 -6196.694,E2 -6196.694} C_VEL
LIN {X 0,Y 495.798,Z 674.558,A -85,B 0,C 180,E1 -6197.982,E2 -6197.982} C_VEL
LIN {X 0,Y 495.603,Z 682.706,A -85,B 0,C 180,E1 -6199.376,E2 -6199.376} C_VEL
LIN {X 0,Y 495.298,Z 690.664,A -85,B 0,C 180,E1 -6201.02,E2 -6201.02} C_VEL
LIN {X 0,Y 495.161,Z 697.001,A -85,B 0,C 180,E1 -6202.661,E2 -6202.661} C_VEL
LIN {X 0,Y 495.089,Z 701.903,A -85,B 0,C 180,E1 -6204.297,E2 -6204.297} C_VEL
LIN {X 0,Y 495.005,Z 705.493,A -85,B 0,C 180,E1 -6205.929,E2 -6205.929} C_VEL
LIN {X 0,Y 495.049,Z 707.865,A -85,B 0,C 180,E1 -6207.559,E2 -6207.559} C_VEL
LIN {X 0,Y 494.907,Z 709.054,A -85,B 0,C 180,E1 -6209.186,E2 -6209.186} C_VEL
LIN {X 0,Y 494.907,Z 709.062,A -85,B 0,C 180,E1 -6210.813,E2 -6210.813} C_VEL
LIN {X 0,Y 495.049,Z 707.889,A -85,B 0,C 180,E1 -6212.441,E2 -6212.441} C_VEL
LIN {X 0,Y 495.004,Z 705.537,A -85,B 0,C 180,E1 -6214.07,E2 -6214.07} C_VEL
LIN {X 0,Y 495.082,Z 701.973,A -85,B 0,C 180,E1 -6215.702,E2 -6215.702} C_VEL
LIN {X 0,Y 495.16,Z 697.098,A -85,B 0,C 180,E1 -6217.339,E2 -6217.339} C_VEL
LIN {X 0,Y 495.298,Z 690.783,A -85,B 0,C 180,E1 -6218.979,E2 -6218.979} C_VEL
LIN {X 0,Y 495.607,Z 682.858,A -85,B 0,C 180,E1 -6220.623,E2 -6220.623} C_VEL
LIN {X 0,Y 495.827,Z 674.642,A -85,B 0,C 180,E1 -6222.034,E2 -6222.034} C_VEL
LIN {X 0,Y 496.357,Z 664.269,A -85,B 0,C 180,E1 -6223.51,E2 -6223.51} C_VEL
LIN {X 0,Y 496.788,Z 653.897,A -85,B 0,C 180,E1 -6224.752,E2 -6224.752} C_VEL
LIN {X 0,Y 497.455,Z 641.585,A -85,B 0,C 180,E1 -6225.985,E2 -6225.985} C_VEL
LIN {X 0,Y 498.005,Z 629.112,A -85,B 0,C 180,E1 -6227.027,E2 -6227.027} C_VEL
LIN {X 0,Y 498.762,Z 615.599,A -85,B 0,C 180,E1 -6227.953,E2 -6227.953} C_VEL
LIN {X 0,Y 499.395,Z 600.647,A -85,B 0,C 180,E1 -6228.779,E2 -6228.779} C_VEL
LIN {X 0,Y 500.004,Z 585.986,A -85,B 0,C 180,E1 -6229.401,E2 -6229.401} C_VEL
LIN {X 0,Y 500.412,Z 571.089,A -85,B 0,C 180,E1 -6229.866,E2 -6229.866} C_VEL
LIN {X 0,Y 500.72,Z 554.95,A -85,B 0,C 180,E1 -6230.193,E2 -6230.193} C_VEL
LIN {X 0,Y 502.05,Z 415.851,A -85,B 0,C 180,E1 -6232.256,E2 -6232.256} C_VEL
LIN {X 0,Y 498.417,Z 395.363,A -85,B 0,C 180,E1 -6232.766,E2 -6232.766} C_VEL
LIN {X 0,Y 499.401,Z 372.152,A -85,B 0,C 180,E1 -6235.755,E2 -6235.755} C_VEL
LIN {X 0,Y 500.005,Z 356.095,A -85,B 0,C 180,E1 -6237.862,E2 -6237.862} C_VEL
LIN {X 0,Y 496.563,Z 341.495,A -85,B 0,C 180,E1 -6240.039,E2 -6240.039} C_VEL
LIN {X 0,Y 495.79,Z 338.355,A -85,B 0,C 180,E1 -6240.535,E2 -6240.535} C_VEL
LIN {X 0,Y 495.756,Z 338.357,A -85,B 0,C 180,E1 -6243.564,E2 -6243.564} C_VEL
LIN {X 0,Y 495.726,Z 338.36,A -85,B 0,C 180,E1 -6246.544,E2 -6246.544} C_VEL
LIN {X 0,Y 495.755,Z 338.355,A -85,B 0,C 180,E1 -6249.638,E2 -6249.638} C_VEL
LIN {X 0,Y 495.738,Z 338.354,A -85,B 0,C 180,E1 -6252.507,E2 -6252.507} C_VEL
LIN {X 0,Y 495.746,Z 338.36,A -85,B 0,C 180,E1 -6255.139,E2 -6255.139} C_VEL
LIN {X 0,Y 495.775,Z 338.349,A -85,B 0,C 180,E1 -6258.221,E2 -6258.221} C_VEL
LIN {X 0,Y 495.748,Z 338.358,A -85,B 0,C 180,E1 -6261.408,E2 -6261.408} C_VEL
LIN {X 0,Y 495.755,Z 338.352,A -85,B 0,C 180,E1 -6264.463,E2 -6264.463} C_VEL
LIN {X 0,Y 495.764,Z 338.355,A -85,B 0,C 180,E1 -6267.406,E2 -6267.406} C_VEL
LIN {X 0,Y 495.763,Z 338.351,A -85,B 0,C 180,E1 -6270.254,E2 -6270.254} C_VEL
LIN {X 0,Y 495.82,Z 338.35,A -85,B 0,C 180,E1 -6273.251,E2 -6273.251} C_VEL
LIN {X 0,Y 495.749,Z 338.353,A -85,B 0,C 180,E1 -6275.725,E2 -6275.725} C_VEL
LIN {X 0,Y 495.744,Z 338.354,A -85,B 0,C 180,E1 -6278.371,E2 -6278.371} C_VEL
LIN {X 0,Y 495.781,Z 338.356,A -85,B 0,C 180,E1 -6280.972,E2 -6280.972} C_VEL
LIN {X 0,Y 495.776,Z 338.351,A -85,B 0,C 180,E1 -6283.53,E2 -6283.53} C_VEL
LIN {X 0,Y 495.794,Z 338.347,A -85,B 0,C 180,E1 -6286.056,E2 -6286.056} C_VEL
LIN {X 0,Y 495.849,Z 338.343,A -85,B 0,C 180,E1 -6288.555,E2 -6288.555} C_VEL
LIN {X 0,Y 495.87,Z 338.337,A -85,B 0,C 180,E1 -6291.852,E2 -6291.852} C_VEL
LIN {X 0,Y 495.887,Z 338.336,A -85,B 0,C 180,E1 -6294.307,E2 -6294.307} C_VEL
LIN {X 0,Y 495.992,Z 338.323,A -85,B 0,C 180,E1 -6297.564,E2 -6297.564} C_VEL
LIN {X 0,Y 495.997,Z 338.321,A -85,B 0,C 180,E1 -6300,E2 -6300} C_VEL
LIN {X 0,Y 495.992,Z 338.325,A -85,B 0,C 180,E1 -6302.437,E2 -6302.437} C_VEL
LIN {X 0,Y 495.896,Z 338.334,A -85,B 0,C 180,E1 -6305.694,E2 -6305.694} C_VEL
LIN {X 0,Y 495.871,Z 338.338,A -85,B 0,C 180,E1 -6308.148,E2 -6308.148} C_VEL
LIN {X 0,Y 495.85,Z 338.341,A -85,B 0,C 180,E1 -6311.446,E2 -6311.446} C_VEL
LIN {X 0,Y 495.788,Z 338.356,A -85,B 0,C 180,E1 -6314.783,E2 -6314.783} C_VEL
LIN {X 0,Y 495.78,Z 338.35,A -85,B 0,C 180,E1 -6317.319,E2 -6317.319} C_VEL
LIN {X 0,Y 495.769,Z 338.35,A -85,B 0,C 180,E1 -6319.891,E2 -6319.891} C_VEL
LIN {X 0,Y 495.758,Z 338.358,A -85,B 0,C 180,E1 -6322.861,E2 -6322.861} C_VEL
LIN {X 0,Y 495.765,Z 338.351,A -85,B 0,C 180,E1 -6326.07,E2 -6326.07} C_VEL
LIN {X 0,Y 495.768,Z 338.357,A -85,B 0,C 180,E1 -6328.815,E2 -6328.815} C_VEL
LIN {X 0,Y 495.754,Z 338.352,A -85,B 0,C 180,E1 -6331.726,E2 -6331.726} C_VEL
LIN {X 0,Y 495.774,Z 338.358,A -85,B 0,C 180,E1 -6334.695,E2 -6334.695} C_VEL
LIN {X 0,Y 495.73,Z 338.355,A -85,B 0,C 180,E1 -6337.562,E2 -6337.562} C_VEL
LIN {X 0,Y 495.753,Z 338.359,A -85,B 0,C 180,E1 -6340.702,E2 -6340.702} C_VEL
LIN {X 0,Y 495.717,Z 338.356,A -85,B 0,C 180,E1 -6343.694,E2 -6343.694} C_VEL
LIN {X 0,Y 495.719,Z 338.361,A -85,B 0,C 180,E1 -6346.307,E2 -6346.307} C_VEL
LIN {X 0,Y 495.754,Z 338.352,A -85,B 0,C 180,E1 -6349.299,E2 -6349.299} C_VEL
LIN {X 0,Y 495.75,Z 338.352,A -85,B 0,C 180,E1 -6351.409,E2 -6351.409} C_VEL
LIN {X 0,Y 495.746,Z 338.361,A -85,B 0,C 180,E1 -6354.463,E2 -6354.463} C_VEL
LIN {X 0,Y 495.769,Z 338.35,A -85,B 0,C 180,E1 -6357.406,E2 -6357.406} C_VEL
LIN {X 0,Y 495.765,Z 338.356,A -85,B 0,C 180,E1 -6360.254,E2 -6360.254} C_VEL
LIN {X 0,Y 495.738,Z 338.355,A -85,B 0,C 180,E1 -6360.759,E2 -6360.759} C_VEL
LIN {X 0,Y 495.066,Z 338.439,A -85,B 0,C 180,E1 -6361.438,E2 -6361.438} C_VEL
LIN {X 0,Y 492.198,Z 338.802,A -85,B 0,C 180,E1 -6362.54,E2 -6362.54} C_VEL
LIN {X 0,Y 489.787,Z 339.099,A -85,B 0,C 180,E1 -6363.428,E2 -6363.428} C_VEL
LIN {X 0,Y 488.771,Z 339.226,A -85,B 0,C 180,E1 -6364.114,E2 -6364.114} C_VEL
LIN {X 0,Y 488.699,Z 339.238,A -85,B 0,C 180,E1 -6364.347,E2 -6364.347} C_VEL
LIN {X 0,Y 488.724,Z 339.228,A -85,B 0,C 180,E1 -6367.154,E2 -6367.154} C_VEL
LIN {X 0,Y 488.726,Z 339.229,A -85,B 0,C 180,E1 -6369.811,E2 -6369.811} C_VEL
LIN {X 0,Y 488.685,Z 339.241,A -85,B 0,C 180,E1 -6372.422,E2 -6372.422} C_VEL
LIN {X 0,Y 488.752,Z 339.225,A -85,B 0,C 180,E1 -6375,E2 -6375} C_VEL
LIN {X 0,Y 488.809,Z 339.225,A -85,B 0,C 180,E1 -6378.388,E2 -6378.388} C_VEL
LIN {X 0,Y 488.765,Z 339.224,A -85,B 0,C 180,E1 -6381.733,E2 -6381.733} C_VEL
LIN {X 0,Y 488.815,Z 339.224,A -85,B 0,C 180,E1 -6384.224,E2 -6384.224} C_VEL
LIN {X 0,Y 488.946,Z 339.2,A -85,B 0,C 180,E1 -6387.529,E2 -6387.529} C_VEL
LIN {X 0,Y 488.945,Z 339.205,A -85,B 0,C 180,E1 -6390,E2 -6390} C_VEL
LIN {X 0,Y 488.945,Z 339.205,A -85,B 0,C 180,E1 -6392.472,E2 -6392.472} C_VEL
LIN {X 0,Y 488.816,Z 339.219,A -85,B 0,C 180,E1 -6395.777,E2 -6395.777} C_VEL
LIN {X 0,Y 488.761,Z 339.231,A -85,B 0,C 180,E1 -6398.268,E2 -6398.268} C_VEL
LIN {X 0,Y 488.788,Z 339.223,A -85,B 0,C 180,E1 -6401.613,E2 -6401.613} C_VEL
LIN {X 0,Y 488.718,Z 339.234,A -85,B 0,C 180,E1 -6405.002,E2 -6405.002} C_VEL
LIN {X 0,Y 488.691,Z 339.242,A -85,B 0,C 180,E1 -6406.018,E2 -6406.018} C_VEL
LIN {X 0,Y 489.794,Z 344.155,A -85,B 0,C 180,E1 -6406.919,E2 -6406.919} C_VEL
LIN {X 0,Y 494.879,Z 357.281,A -85,B 0,C 180,E1 -6407.381,E2 -6407.381} C_VEL
LIN {X 0,Y 495.644,Z 360.577,A -85,B 0,C 180,E1 -6407.47,E2 -6407.47} C_VEL
LIN {X 0,Y 494.126,Z 508.586,A -85,B 0,C 180,E1 -6409.73,E2 -6409.73} C_VEL
LIN {X 0,Y 493.774,Z 523.835,A -85,B 0,C 180,E1 -6410.127,E2 -6410.127} C_VEL
LIN {X 0,Y 493.346,Z 538.654,A -85,B 0,C 180,E1 -6410.684,E2 -6410.684} C_VEL
LIN {X 0,Y 492.725,Z 553.773,A -85,B 0,C 180,E1 -6411.439,E2 -6411.439} C_VEL
LIN {X 0,Y 492.067,Z 567.627,A -85,B 0,C 180,E1 -6412.318,E2 -6412.318} C_VEL
LIN {X 0,Y 491.42,Z 579.922,A -85,B 0,C 180,E1 -6413.271,E2 -6413.271} C_VEL
LIN {X 0,Y 490.685,Z 592.21,A -85,B 0,C 180,E1 -6414.418,E2 -6414.418} C_VEL
LIN {X 0,Y 490.073,Z 603.683,A -85,B 0,C 180,E1 -6415.71,E2 -6415.71} C_VEL
LIN {X 0,Y 489.448,Z 613.958,A -85,B 0,C 180,E1 -6417.093,E2 -6417.093} C_VEL
LIN {X 0,Y 489.015,Z 622.802,A -85,B 0,C 180,E1 -6418.523,E2 -6418.523} C_VEL
LIN {X 0,Y 488.597,Z 630.371,A -85,B 0,C 180,E1 -6419.99,E2 -6419.99} C_VEL
LIN {X 0,Y 488.366,Z 636.947,A -85,B 0,C 180,E1 -6421.541,E2 -6421.541} C_VEL
LIN {X 0,Y 488.121,Z 642.485,A -85,B 0,C 180,E1 -6423.17,E2 -6423.17} C_VEL
LIN {X 0,Y 487.977,Z 646.775,A -85,B 0,C 180,E1 -6424.821,E2 -6424.821} C_VEL
LIN {X 0,Y 487.856,Z 649.46,A -85,B 0,C 180,E1 -6426.222,E2 -6426.222} C_VEL
LIN {X 0,Y 487.819,Z 651.236,A -85,B 0,C 180,E1 -6427.59,E2 -6427.59} C_VEL
LIN {X 0,Y 487.807,Z 652.398,A -85,B 0,C 180,E1 -6429.34,E2 -6429.34} C_VEL
LIN {X 0,Y 487.799,Z 652.469,A -85,B 0,C 180,E1 -6430.417,E2 -6430.417} C_VEL
LIN {X 0,Y 487.844,Z 652.068,A -85,B 0,C 180,E1 -6431.506,E2 -6431.506} C_VEL
LIN {X 0,Y 487.865,Z 651.074,A -85,B 0,C 180,E1 -6432.719,E2 -6432.719} C_VEL
LIN {X 0,Y 487.914,Z 649.423,A -85,B 0,C 180,E1 -6433.928,E2 -6433.928} C_VEL
LIN {X 0,Y 488.065,Z 646.088,A -85,B 0,C 180,E1 -6435.617,E2 -6435.617} C_VEL
LIN {X 0,Y 488.193,Z 641.073,A -85,B 0,C 180,E1 -6437.42,E2 -6437.42} C_VEL
LIN {X 0,Y 488.424,Z 634.948,A -85,B 0,C 180,E1 -6439.102,E2 -6439.102} C_VEL
LIN {X 0,Y 488.76,Z 627.399,A -85,B 0,C 180,E1 -6440.751,E2 -6440.751} C_VEL
LIN {X 0,Y 489.211,Z 619.329,A -85,B 0,C 180,E1 -6442.198,E2 -6442.198} C_VEL
LIN {X 0,Y 489.663,Z 610.727,A -85,B 0,C 180,E1 -6443.49,E2 -6443.49} C_VEL
LIN {X 0,Y 490.268,Z 600.455,A -85,B 0,C 180,E1 -6444.796,E2 -6444.796} C_VEL
LIN {X 0,Y 491.006,Z 588.469,A -85,B 0,C 180,E1 -6446.066,E2 -6446.066} C_VEL
LIN {X 0,Y 491.596,Z 576.872,A -85,B 0,C 180,E1 -6447.094,E2 -6447.094} C_VEL
LIN {X 0,Y 492.202,Z 564.551,A -85,B 0,C 180,E1 -6448.005,E2 -6448.005} C_VEL
LIN {X 0,Y 492.91,Z 551.071,A -85,B 0,C 180,E1 -6448.815,E2 -6448.815} C_VEL
LIN {X 0,Y 493.348,Z 538.124,A -85,B 0,C 180,E1 -6449.443,E2 -6449.443} C_VEL
LIN {X 0,Y 493.808,Z 523.205,A -85,B 0,C 180,E1 -6449.991,E2 -6449.991} C_VEL
LIN {X 0,Y 494.121,Z 507.903,A -85,B 0,C 180,E1 -6450.379,E2 -6450.379} C_VEL
LIN {X 0,Y 495.704,Z 360.605,A -85,B 0,C 180,E1 -6452.636,E2 -6452.636} C_VEL
LIN {X 0,Y 494.078,Z 354.96,A -85,B 0,C 180,E1 -6452.808,E2 -6452.808} C_VEL
LIN {X 0,Y 489.993,Z 344.904,A -85,B 0,C 180,E1 -6453.197,E2 -6453.197} C_VEL
LIN {X 0,Y 488.7,Z 339.237,A -85,B 0,C 180,E1 -6454.327,E2 -6454.327} C_VEL
LIN {X 0,Y 488.711,Z 339.234,A -85,B 0,C 180,E1 -6457.152,E2 -6457.152} C_VEL
LIN {X 0,Y 488.714,Z 339.237,A -85,B 0,C 180,E1 -6459.81,E2 -6459.81} C_VEL
LIN {X 0,Y 488.685,Z 339.233,A -85,B 0,C 180,E1 -6462.421,E2 -6462.421} C_VEL
LIN {X 0,Y 488.752,Z 339.227,A -85,B 0,C 180,E1 -6464.999,E2 -6464.999} C_VEL
LIN {X 0,Y 488.808,Z 339.22,A -85,B 0,C 180,E1 -6468.387,E2 -6468.387} C_VEL
LIN {X 0,Y 488.764,Z 339.231,A -85,B 0,C 180,E1 -6471.732,E2 -6471.732} C_VEL
LIN {X 0,Y 488.817,Z 339.219,A -85,B 0,C 180,E1 -6474.223,E2 -6474.223} C_VEL
LIN {X 0,Y 488.947,Z 339.206,A -85,B 0,C 180,E1 -6477.528,E2 -6477.528} C_VEL
LIN {X 0,Y 488.971,Z 339.201,A -85,B 0,C 180,E1 -6480,E2 -6480} C_VEL
LIN {X 0,Y 488.956,Z 339.199,A -85,B 0,C 180,E1 -6482.471,E2 -6482.471} C_VEL
LIN {X 0,Y 488.832,Z 339.219,A -85,B 0,C 180,E1 -6485.776,E2 -6485.776} C_VEL
LIN {X 0,Y 488.782,Z 339.222,A -85,B 0,C 180,E1 -6488.267,E2 -6488.267} C_VEL
LIN {X 0,Y 488.808,Z 339.222,A -85,B 0,C 180,E1 -6491.612,E2 -6491.612} C_VEL
LIN {X 0,Y 488.763,Z 339.228,A -85,B 0,C 180,E1 -6495,E2 -6495} C_VEL
LIN {X 0,Y 488.749,Z 339.224,A -85,B 0,C 180,E1 -6498.442,E2 -6498.442} C_VEL
LIN {X 0,Y 488.709,Z 339.236,A -85,B 0,C 180,E1 -6501.07,E2 -6501.07} C_VEL
LIN {X 0,Y 488.686,Z 339.233,A -85,B 0,C 180,E1 -6503.746,E2 -6503.746} C_VEL
LIN {X 0,Y 488.794,Z 339.225,A -85,B 0,C 180,E1 -6506.943,E2 -6506.943} C_VEL
LIN {X 0,Y 488.711,Z 339.229,A -85,B 0,C 180,E1 -6510.362,E2 -6510.362} C_VEL
LIN {X 0,Y 488.736,Z 339.231,A -85,B 0,C 180,E1 -6513.484,E2 -6513.484} C_VEL
LIN {X 0,Y 488.684,Z 339.236,A -85,B 0,C 180,E1 -6516.354,E2 -6516.354} C_VEL
LIN {X 0,Y 488.703,Z 339.237,A -85,B 0,C 180,E1 -6519.254,E2 -6519.254} C_VEL
LIN {X 0,Y 488.71,Z 339.233,A -85,B 0,C 180,E1 -6521.6,E2 -6521.6} C_VEL
LIN {X 0,Y 488.714,Z 339.236,A -85,B 0,C 180,E1 -6524.801,E2 -6524.801} C_VEL
LIN {X 0,Y 488.696,Z 339.235,A -85,B 0,C 180,E1 -6527.475,E2 -6527.475} C_VEL
LIN {X 0,Y 488.734,Z 339.231,A -85,B 0,C 180,E1 -6529.676,E2 -6529.676} C_VEL
LIN {X 0,Y 488.681,Z 339.239,A -85,B 0,C 180,E1 -6532.841,E2 -6532.841} C_VEL
LIN {X 0,Y 488.731,Z 339.231,A -85,B 0,C 180,E1 -6535.887,E2 -6535.887} C_VEL
LIN {X 0,Y 488.724,Z 339.267,A -85,B 0,C 180,E1 -6539.294,E2 -6539.294} C_VEL
LIN {X 0,Y 492.51,Z 354.755,A -85,B 0,C 180,E1 -6541.675,E2 -6541.675} C_VEL
LIN {X 0,Y 493.025,Z 358.867,A -85,B 0,C 180,E1 -6542.262,E2 -6542.262} C_VEL
LIN {X 0,Y 492.036,Z 380.193,A -85,B 0,C 180,E1 -6545.079,E2 -6545.079} C_VEL
LIN {X 0,Y 491.479,Z 394.227,A -85,B 0,C 180,E1 -6546.907,E2 -6546.907} C_VEL
LIN {X 0,Y 495.408,Z 416.425,A -85,B 0,C 180,E1 -6547.456,E2 -6547.456} C_VEL
LIN {X 0,Y 493.895,Z 562.061,A -85,B 0,C 180,E1 -6549.678,E2 -6549.678} C_VEL
LIN {X 0,Y 493.427,Z 578.159,A -85,B 0,C 180,E1 -6550.097,E2 -6550.097} C_VEL
LIN {X 0,Y 492.899,Z 591.849,A -85,B 0,C 180,E1 -6550.603,E2 -6550.603} C_VEL
LIN {X 0,Y 492.314,Z 605.555,A -85,B 0,C 180,E1 -6551.264,E2 -6551.264} C_VEL
LIN {X 0,Y 491.611,Z 619.38,A -85,B 0,C 180,E1 -6552.099,E2 -6552.099} C_VEL
LIN {X 0,Y 490.945,Z 632.1,A -85,B 0,C 180,E1 -6553.041,E2 -6553.041} C_VEL
LIN {X 0,Y 490.291,Z 645.014,A -85,B 0,C 180,E1 -6554.195,E2 -6554.195} C_VEL
LIN {X 0,Y 489.601,Z 656.735,A -85,B 0,C 180,E1 -6555.451,E2 -6555.451} C_VEL
LIN {X 0,Y 489.16,Z 666.612,A -85,B 0,C 180,E1 -6556.71,E2 -6556.71} C_VEL
LIN {X 0,Y 488.691,Z 675.706,A -85,B 0,C 180,E1 -6558.075,E2 -6558.075} C_VEL
LIN {X 0,Y 488.487,Z 683.359,A -85,B 0,C 180,E1 -6559.43,E2 -6559.43} C_VEL
LIN {X 0,Y 488.232,Z 690.215,A -85,B 0,C 180,E1 -6560.889,E2 -6560.889} C_VEL
LIN {X 0,Y 488.065,Z 696.562,A -85,B 0,C 180,E1 -6562.553,E2 -6562.553} C_VEL
LIN {X 0,Y 487.986,Z 701.474,A -85,B 0,C 180,E1 -6564.214,E2 -6564.214} C_VEL
LIN {X 0,Y 487.908,Z 705.072,A -85,B 0,C 180,E1 -6565.87,E2 -6565.87} C_VEL
LIN {X 0,Y 487.984,Z 707.451,A -85,B 0,C 180,E1 -6567.523,E2 -6567.523} C_VEL
LIN {X 0,Y 487.83,Z 708.644,A -85,B 0,C 180,E1 -6569.174,E2 -6569.174} C_VEL
LIN {X 0,Y 487.83,Z 708.656,A -85,B 0,C 180,E1 -6570.825,E2 -6570.825} C_VEL
LIN {X 0,Y 487.967,Z 707.483,A -85,B 0,C 180,E1 -6572.476,E2 -6572.476} C_VEL
LIN {X 0,Y 487.906,Z 705.13,A -85,B 0,C 180,E1 -6574.13,E2 -6574.13} C_VEL
LIN {X 0,Y 487.98,Z 701.563,A -85,B 0,C 180,E1 -6575.786,E2 -6575.786} C_VEL
LIN {X 0,Y 488.064,Z 696.684,A -85,B 0,C 180,E1 -6577.446,E2 -6577.446} C_VEL
LIN {X 0,Y 488.231,Z 690.365,A -85,B 0,C 180,E1 -6579.11,E2 -6579.11} C_VEL
LIN {X 0,Y 488.567,Z 682.435,A -85,B 0,C 180,E1 -6580.778,E2 -6580.778} C_VEL
LIN {X 0,Y 488.797,Z 674.272,A -85,B 0,C 180,E1 -6582.2,E2 -6582.2} C_VEL
LIN {X 0,Y 489.333,Z 663.826,A -85,B 0,C 180,E1 -6583.708,E2 -6583.708} C_VEL
LIN {X 0,Y 489.848,Z 653.451,A -85,B 0,C 180,E1 -6584.966,E2 -6584.966} C_VEL
LIN {X 0,Y 490.495,Z 642.057,A -85,B 0,C 180,E1 -6586.128,E2 -6586.128} C_VEL
LIN {X 0,Y 491.155,Z 628.644,A -85,B 0,C 180,E1 -6587.272,E2 -6587.272} C_VEL
LIN {X 0,Y 491.919,Z 615.112,A -85,B 0,C 180,E1 -6588.211,E2 -6588.211} C_VEL
LIN {X 0,Y 492.608,Z 600.131,A -85,B 0,C 180,E1 -6589.047,E2 -6589.047} C_VEL
LIN {X 0,Y 493.276,Z 584.904,A -85,B 0,C 180,E1 -6589.696,E2 -6589.696} C_VEL
LIN {X 0,Y 493.737,Z 569.798,A -85,B 0,C 180,E1 -6590.165,E2 -6590.165} C_VEL
LIN {X 0,Y 494.047,Z 554.15,A -85,B 0,C 180,E1 -6590.478,E2 -6590.478} C_VEL
LIN {X 0,Y 495.472,Z 417.28,A -85,B 0,C 180,E1 -6592.537,E2 -6592.537} C_VEL
LIN {X 0,Y 491.568,Z 394.978,A -85,B 0,C 180,E1 -6593.101,E2 -6593.101} C_VEL
LIN {X 0,Y 492.591,Z 372.844,A -85,B 0,C 180,E1 -6595.993,E2 -6595.993} C_VEL
LIN {X 0,Y 493.243,Z 358.151,A -85,B 0,C 180,E1 -6597.944,E2 -6597.944} C_VEL
LIN {X 0,Y 489.848,Z 343.62,A -85,B 0,C 180,E1 -6600.142,E2 -6600.142} C_VEL
LIN {X 0,Y 488.721,Z 339.234,A -85,B 0,C 180,E1 -6600.86,E2 -6600.86} C_VEL
LIN {X 0,Y 488.728,Z 339.231,A -85,B 0,C 180,E1 -6604.113,E2 -6604.113} C_VEL
LIN {X 0,Y 488.677,Z 339.242,A -85,B 0,C 180,E1 -6607.159,E2 -6607.159} C_VEL
LIN {X 0,Y 488.715,Z 339.228,A -85,B 0,C 180,E1 -6610.344,E2 -6610.344} C_VEL
LIN {X 0,Y 488.713,Z 339.232,A -85,B 0,C 180,E1 -6612.827,E2 -6612.827} C_VEL
LIN {X 0,Y 488.699,Z 339.231,A -85,B 0,C 180,E1 -6615.976,E2 -6615.976} C_VEL
LIN {X 0,Y 488.716,Z 339.23,A -85,B 0,C 180,E1 -6618.586,E2 -6618.586} C_VEL
LIN {X 0,Y 488.677,Z 339.234,A -85,B 0,C 180,E1 -6621.8,E2 -6621.8} C_VEL
LIN {X 0,Y 488.726,Z 339.234,A -85,B 0,C 180,E1 -6625.051,E2 -6625.051} C_VEL
LIN {X 0,Y 488.7,Z 339.23,A -85,B 0,C 180,E1 -6628.046,E2 -6628.046} C_VEL
LIN {X 0,Y 488.72,Z 339.231,A -85,B 0,C 180,E1 -6630.73,E2 -6630.73} C_VEL
LIN {X 0,Y 488.753,Z 339.227,A -85,B 0,C 180,E1 -6633.528,E2 -6633.528} C_VEL
LIN {X 0,Y 488.691,Z 339.232,A -85,B 0,C 180,E1 -6636.255,E2 -6636.255} C_VEL
LIN {X 0,Y 488.743,Z 339.232,A -85,B 0,C 180,E1 -6639.176,E2 -6639.176} C_VEL
LIN {X 0,Y 488.756,Z 339.225,A -85,B 0,C 180,E1 -6641.628,E2 -6641.628} C_VEL
LIN {X 0,Y 488.759,Z 339.232,A -85,B 0,C 180,E1 -6645,E2 -6645} C_VEL
LIN {X 0,Y 488.803,Z 339.219,A -85,B 0,C 180,E1 -6648.388,E2 -6648.388} C_VEL
LIN {X 0,Y 488.815,Z 339.217,A -85,B 0,C 180,E1 -6651.734,E2 -6651.734} C_VEL
LIN {X 0,Y 488.845,Z 339.213,A -85,B 0,C 180,E1 -6654.224,E2 -6654.224} C_VEL
LIN {X 0,Y 488.959,Z 339.199,A -85,B 0,C 180,E1 -6657.529,E2 -6657.529} C_VEL
LIN {X 0,Y 488.952,Z 339.207,A -85,B 0,C 180,E1 -6660.824,E2 -6660.824} C_VEL
LIN {X 0,Y 488.959,Z 339.201,A -85,B 0,C 180,E1 -6662.472,E2 -6662.472} C_VEL
LIN {X 0,Y 488.855,Z 339.211,A -85,B 0,C 180,E1 -6665.776,E2 -6665.776} C_VEL
LIN {X 0,Y 488.816,Z 339.218,A -85,B 0,C 180,E1 -6668.267,E2 -6668.267} C_VEL
LIN {X 0,Y 488.804,Z 339.218,A -85,B 0,C 180,E1 -6671.613,E2 -6671.613} C_VEL
LIN {X 0,Y 488.76,Z 339.229,A -85,B 0,C 180,E1 -6675.001,E2 -6675.001} C_VEL
LIN {X 0,Y 488.753,Z 339.228,A -85,B 0,C 180,E1 -6678.443,E2 -6678.443} C_VEL
LIN {X 0,Y 488.705,Z 339.234,A -85,B 0,C 180,E1 -6681.071,E2 -6681.071} C_VEL
LIN {X 0,Y 488.686,Z 339.232,A -85,B 0,C 180,E1 -6683.746,E2 -6683.746} C_VEL
LIN {X 0,Y 488.736,Z 339.231,A -85,B 0,C 180,E1 -6686.474,E2 -6686.474} C_VEL
LIN {X 0,Y 488.721,Z 339.229,A -85,B 0,C 180,E1 -6689.271,E2 -6689.271} C_VEL
LIN {X 0,Y 488.702,Z 339.232,A -85,B 0,C 180,E1 -6692.148,E2 -6692.148} C_VEL
LIN {X 0,Y 488.721,Z 339.23,A -85,B 0,C 180,E1 -6695.115,E2 -6695.115} C_VEL
LIN {X 0,Y 488.68,Z 339.236,A -85,B 0,C 180,E1 -6698.201,E2 -6698.201} C_VEL
LIN {X 0,Y 488.718,Z 339.233,A -85,B 0,C 180,E1 -6700.345,E2 -6700.345} C_VEL
LIN {X 0,Y 488.676,Z 339.233,A -85,B 0,C 180,E1 -6703.656,E2 -6703.656} C_VEL
LIN {X 0,Y 488.678,Z 339.238,A -85,B 0,C 180,E1 -6706.345,E2 -6706.345} C_VEL
LIN {X 0,Y 488.704,Z 339.23,A -85,B 0,C 180,E1 -6709.674,E2 -6709.674} C_VEL
LIN {X 0,Y 488.671,Z 339.238,A -85,B 0,C 180,E1 -6712.841,E2 -6712.841} C_VEL
LIN {X 0,Y 488.731,Z 339.228,A -85,B 0,C 180,E1 -6715.888,E2 -6715.888} C_VEL
LIN {X 0,Y 488.693,Z 339.235,A -85,B 0,C 180,E1 -6718.821,E2 -6718.821} C_VEL
LIN {X 0,Y 488.713,Z 339.229,A -85,B 0,C 180,E1 -6721.67,E2 -6721.67} C_VEL
LIN {X 0,Y 488.699,Z 339.238,A -85,B 0,C 180,E1 -6724.347,E2 -6724.347} C_VEL
LIN {X 0,Y 488.058,Z 339.325,A -85,B 0,C 180,E1 -6725.035,E2 -6725.035} C_VEL
LIN {X 0,Y 485.207,Z 339.677,A -85,B 0,C 180,E1 -6726.152,E2 -6726.152} C_VEL
LIN {X 0,Y 482.775,Z 339.972,A -85,B 0,C 180,E1 -6727.052,E2 -6727.052} C_VEL
LIN {X 0,Y 481.725,Z 340.1,A -85,B 0,C 180,E1 -6727.748,E2 -6727.748} C_VEL
LIN {X 0,Y 481.637,Z 340.111,A -85,B 0,C 180,E1 -6727.983,E2 -6727.983} C_VEL
LIN {X 0,Y 481.703,Z 340.111,A -85,B 0,C 180,E1 -6730.393,E2 -6730.393} C_VEL
LIN {X 0,Y 481.625,Z 340.113,A -85,B 0,C 180,E1 -6733.032,E2 -6733.032} C_VEL
LIN {X 0,Y 481.68,Z 340.105,A -85,B 0,C 180,E1 -6735.639,E2 -6735.639} C_VEL
LIN {X 0,Y 481.754,Z 340.102,A -85,B 0,C 180,E1 -6738.216,E2 -6738.216} C_VEL
LIN {X 0,Y 481.724,Z 340.1,A -85,B 0,C 180,E1 -6741.611,E2 -6741.611} C_VEL
LIN {X 0,Y 481.776,Z 340.099,A -85,B 0,C 180,E1 -6744.139,E2 -6744.139} C_VEL
LIN {X 0,Y 481.911,Z 340.076,A -85,B 0,C 180,E1 -6747.493,E2 -6747.493} C_VEL
LIN {X 0,Y 481.914,Z 340.081,A -85,B 0,C 180,E1 -6750,E2 -6750} C_VEL
LIN {X 0,Y 481.91,Z 340.081,A -85,B 0,C 180,E1 -6752.508,E2 -6752.508} C_VEL
LIN {X 0,Y 481.778,Z 340.096,A -85,B 0,C 180,E1 -6755.861,E2 -6755.861} C_VEL
LIN {X 0,Y 481.72,Z 340.106,A -85,B 0,C 180,E1 -6758.389,E2 -6758.389} C_VEL
LIN {X 0,Y 481.739,Z 340.102,A -85,B 0,C 180,E1 -6761.786,E2 -6761.786} C_VEL
LIN {X 0,Y 481.69,Z 340.11,A -85,B 0,C 180,E1 -6765.226,E2 -6765.226} C_VEL
LIN {X 0,Y 481.668,Z 340.235,A -85,B 0,C 180,E1 -6765.767,E2 -6765.767} C_VEL
LIN {X 0,Y 482.546,Z 344.298,A -85,B 0,C 180,E1 -6766.548,E2 -6766.548} C_VEL
LIN {X 0,Y 488.538,Z 359.284,A -85,B 0,C 180,E1 -6767.098,E2 -6767.098} C_VEL
LIN {X 0,Y 489.137,Z 362.784,A -85,B 0,C 180,E1 -6767.185,E2 -6767.185} C_VEL
LIN {X 0,Y 487.46,Z 508.847,A -85,B 0,C 180,E1 -6769.445,E2 -6769.445} C_VEL
LIN {X 0,Y 487.11,Z 524.195,A -85,B 0,C 180,E1 -6769.85,E2 -6769.85} C_VEL
LIN {X 0,Y 486.651,Z 538.47,A -85,B 0,C 180,E1 -6770.39,E2 -6770.39} C_VEL
LIN {X 0,Y 486.009,Z 553.452,A -85,B 0,C 180,E1 -6771.138,E2 -6771.138} C_VEL
LIN {X 0,Y 485.302,Z 567.777,A -85,B 0,C 180,E1 -6772.053,E2 -6772.053} C_VEL
LIN {X 0,Y 484.583,Z 580.517,A -85,B 0,C 180,E1 -6773.054,E2 -6773.054} C_VEL
LIN {X 0,Y 483.807,Z 592.889,A -85,B 0,C 180,E1 -6774.229,E2 -6774.229} C_VEL
LIN {X 0,Y 483.137,Z 604.735,A -85,B 0,C 180,E1 -6775.591,E2 -6775.591} C_VEL
LIN {X 0,Y 482.443,Z 615.363,A -85,B 0,C 180,E1 -6777.065,E2 -6777.065} C_VEL
LIN {X 0,Y 481.982,Z 624.126,A -85,B 0,C 180,E1 -6778.525,E2 -6778.525} C_VEL
LIN {X 0,Y 481.564,Z 632.124,A -85,B 0,C 180,E1 -6780.14,E2 -6780.14} C_VEL
LIN {X 0,Y 481.283,Z 638.461,A -85,B 0,C 180,E1 -6781.715,E2 -6781.715} C_VEL
LIN {X 0,Y 481.069,Z 643.145,A -85,B 0,C 180,E1 -6783.163,E2 -6783.163} C_VEL
LIN {X 0,Y 480.921,Z 647.171,A -85,B 0,C 180,E1 -6784.746,E2 -6784.746} C_VEL
LIN {X 0,Y 480.772,Z 650.338,A -85,B 0,C 180,E1 -6786.486,E2 -6786.486} C_VEL
LIN {X 0,Y 480.733,Z 651.95,A -85,B 0,C 180,E1 -6787.881,E2 -6787.881} C_VEL
LIN {X 0,Y 480.718,Z 652.781,A -85,B 0,C 180,E1 -6789.208,E2 -6789.208} C_VEL
LIN {X 0,Y 480.726,Z 652.863,A -85,B 0,C 180,E1 -6790.516,E2 -6790.516} C_VEL
LIN {X 0,Y 480.748,Z 651.949,A -85,B 0,C 180,E1 -6792.258,E2 -6792.258} C_VEL
LIN {X 0,Y 480.818,Z 650.689,A -85,B 0,C 180,E1 -6793.393,E2 -6793.393} C_VEL
LIN {X 0,Y 480.892,Z 648.881,A -85,B 0,C 180,E1 -6794.548,E2 -6794.548} C_VEL
LIN {X 0,Y 481.033,Z 645.304,A -85,B 0,C 180,E1 -6796.18,E2 -6796.18} C_VEL
LIN {X 0,Y 481.197,Z 640.612,A -85,B 0,C 180,E1 -6797.79,E2 -6797.79} C_VEL
LIN {X 0,Y 481.428,Z 634.717,A -85,B 0,C 180,E1 -6799.386,E2 -6799.386} C_VEL
LIN {X 0,Y 481.787,Z 627.822,A -85,B 0,C 180,E1 -6800.903,E2 -6800.903} C_VEL
LIN {X 0,Y 482.223,Z 620.417,A -85,B 0,C 180,E1 -6802.257,E2 -6802.257} C_VEL
LIN {X 0,Y 482.7,Z 611.673,A -85,B 0,C 180,E1 -6803.607,E2 -6803.607} C_VEL
LIN {X 0,Y 483.361,Z 601.362,A -85,B 0,C 180,E1 -6804.947,E2 -6804.947} C_VEL
LIN {X 0,Y 484.122,Z 589.873,A -85,B 0,C 180,E1 -6806.195,E2 -6806.195} C_VEL
LIN {X 0,Y 484.794,Z 577.348,A -85,B 0,C 180,E1 -6807.331,E2 -6807.331} C_VEL
LIN {X 0,Y 485.515,Z 564.242,A -85,B 0,C 180,E1 -6808.307,E2 -6808.307} C_VEL
LIN {X 0,Y 486.161,Z 550.734,A -85,B 0,C 180,E1 -6809.123,E2 -6809.123} C_VEL
LIN {X 0,Y 486.786,Z 535.953,A -85,B 0,C 180,E1 -6809.821,E2 -6809.821} C_VEL
LIN {X 0,Y 487.205,Z 520.339,A -85,B 0,C 180,E1 -6810.368,E2 -6810.368} C_VEL
LIN {X 0,Y 487.537,Z 504.652,A -85,B 0,C 180,E1 -6810.73,E2 -6810.73} C_VEL
LIN {X 0,Y 489.193,Z 361.767,A -85,B 0,C 180,E1 -6812.947,E2 -6812.947} C_VEL
LIN {X 0,Y 487.477,Z 356.519,A -85,B 0,C 180,E1 -6813.121,E2 -6813.121} C_VEL
LIN {X 0,Y 482.888,Z 345.416,A -85,B 0,C 180,E1 -6813.559,E2 -6813.559} C_VEL
LIN {X 0,Y 481.654,Z 340.114,A -85,B 0,C 180,E1 -6814.634,E2 -6814.634} C_VEL
LIN {X 0,Y 481.639,Z 340.117,A -85,B 0,C 180,E1 -6817.704,E2 -6817.704} C_VEL
LIN {X 0,Y 481.694,Z 340.105,A -85,B 0,C 180,E1 -6820.392,E2 -6820.392} C_VEL
LIN {X 0,Y 481.625,Z 340.112,A -85,B 0,C 180,E1 -6823.031,E2 -6823.031} C_VEL
LIN {X 0,Y 481.682,Z 340.114,A -85,B 0,C 180,E1 -6825.638,E2 -6825.638} C_VEL
LIN {X 0,Y 481.754,Z 340.1,A -85,B 0,C 180,E1 -6828.215,E2 -6828.215} C_VEL
LIN {X 0,Y 481.723,Z 340.107,A -85,B 0,C 180,E1 -6831.611,E2 -6831.611} C_VEL
LIN {X 0,Y 481.778,Z 340.096,A -85,B 0,C 180,E1 -6834.139,E2 -6834.139} C_VEL
LIN {X 0,Y 481.912,Z 340.082,A -85,B 0,C 180,E1 -6837.492,E2 -6837.492} C_VEL
LIN {X 0,Y 481.941,Z 340.077,A -85,B 0,C 180,E1 -6840,E2 -6840} C_VEL
LIN {X 0,Y 481.922,Z 340.076,A -85,B 0,C 180,E1 -6842.507,E2 -6842.507} C_VEL
LIN {X 0,Y 481.791,Z 340.096,A -85,B 0,C 180,E1 -6845.86,E2 -6845.86} C_VEL
LIN {X 0,Y 481.738,Z 340.099,A -85,B 0,C 180,E1 -6848.388,E2 -6848.388} C_VEL
LIN {X 0,Y 481.753,Z 340.099,A -85,B 0,C 180,E1 -6851.785,E2 -6851.785} C_VEL
LIN {X 0,Y 481.744,Z 340.103,A -85,B 0,C 180,E1 -6855.224,E2 -6855.224} C_VEL
LIN {X 0,Y 481.711,Z 340.102,A -85,B 0,C 180,E1 -6858.721,E2 -6858.721} C_VEL
LIN {X 0,Y 481.648,Z 340.114,A -85,B 0,C 180,E1 -6861.394,E2 -6861.394} C_VEL
LIN {X 0,Y 481.672,Z 340.105,A -85,B 0,C 180,E1 -6864.113,E2 -6864.113} C_VEL
LIN {X 0,Y 481.749,Z 340.102,A -85,B 0,C 180,E1 -6867.139,E2 -6867.139} C_VEL
LIN {X 0,Y 481.681,Z 340.106,A -85,B 0,C 180,E1 -6869.741,E2 -6869.741} C_VEL
LIN {X 0,Y 481.674,Z 340.109,A -85,B 0,C 180,E1 -6872.674,E2 -6872.674} C_VEL
LIN {X 0,Y 481.638,Z 340.114,A -85,B 0,C 180,E1 -6875.709,E2 -6875.709} C_VEL
LIN {X 0,Y 481.672,Z 340.114,A -85,B 0,C 180,E1 -6878.859,E2 -6878.859} C_VEL
LIN {X 0,Y 481.655,Z 340.111,A -85,B 0,C 180,E1 -6881.913,E2 -6881.913} C_VEL
LIN {X 0,Y 481.661,Z 340.112,A -85,B 0,C 180,E1 -6884.457,E2 -6884.457} C_VEL
LIN {X 0,Y 481.655,Z 340.111,A -85,B 0,C 180,E1 -6887.84,E2 -6887.84} C_VEL
LIN {X 0,Y 481.682,Z 340.111,A -85,B 0,C 180,E1 -6890.651,E2 -6890.651} C_VEL
LIN {X 0,Y 481.628,Z 340.116,A -85,B 0,C 180,E1 -6893.376,E2 -6893.376} C_VEL
LIN {X 0,Y 481.711,Z 340.108,A -85,B 0,C 180,E1 -6896.33,E2 -6896.33} C_VEL
LIN {X 0,Y 481.701,Z 340.265,A -85,B 0,C 180,E1 -6898.989,E2 -6898.989} C_VEL
LIN {X 0,Y 485.606,Z 356.085,A -85,B 0,C 180,E1 -6901.471,E2 -6901.471} C_VEL
LIN {X 0,Y 486.153,Z 358.692,A -85,B 0,C 180,E1 -6901.865,E2 -6901.865} C_VEL
LIN {X 0,Y 485.697,Z 371.846,A -85,B 0,C 180,E1 -6903.65,E2 -6903.65} C_VEL
LIN {X 0,Y 484.639,Z 393.648,A -85,B 0,C 180,E1 -6906.543,E2 -6906.543} C_VEL
LIN {X 0,Y 488.871,Z 417.597,A -85,B 0,C 180,E1 -6907.16,E2 -6907.16} C_VEL
LIN {X 0,Y 487.2,Z 561.379,A -85,B 0,C 180,E1 -6909.386,E2 -6909.386} C_VEL
LIN {X 0,Y 486.741,Z 577.362,A -85,B 0,C 180,E1 -6909.805,E2 -6909.805} C_VEL
LIN {X 0,Y 486.161,Z 591.658,A -85,B 0,C 180,E1 -6910.34,E2 -6910.34} C_VEL
LIN {X 0,Y 485.447,Z 606.936,A -85,B 0,C 180,E1 -6911.099,E2 -6911.099} C_VEL
LIN {X 0,Y 484.698,Z 620.425,A -85,B 0,C 180,E1 -6911.945,E2 -6911.945} C_VEL
LIN {X 0,Y 483.909,Z 634.168,A -85,B 0,C 180,E1 -6913.005,E2 -6913.005} C_VEL
LIN {X 0,Y 483.258,Z 646.662,A -85,B 0,C 180,E1 -6914.176,E2 -6914.176} C_VEL
LIN {X 0,Y 482.547,Z 658.051,A -85,B 0,C 180,E1 -6915.449,E2 -6915.449} C_VEL
LIN {X 0,Y 482.006,Z 669.132,A -85,B 0,C 180,E1 -6916.938,E2 -6916.938} C_VEL
LIN {X 0,Y 481.589,Z 678.346,A -85,B 0,C 180,E1 -6918.424,E2 -6918.424} C_VEL
LIN {X 0,Y 481.257,Z 685.989,A -85,B 0,C 180,E1 -6919.907,E2 -6919.907} C_VEL
LIN {X 0,Y 481.057,Z 693.135,A -85,B 0,C 180,E1 -6921.599,E2 -6921.599} C_VEL
LIN {X 0,Y 480.956,Z 698.757,A -85,B 0,C 180,E1 -6923.286,E2 -6923.286} C_VEL
LIN {X 0,Y 480.855,Z 703.007,A -85,B 0,C 180,E1 -6924.969,E2 -6924.969} C_VEL
LIN {X 0,Y 480.873,Z 705.995,A -85,B 0,C 180,E1 -6926.648,E2 -6926.648} C_VEL
LIN {X 0,Y 480.822,Z 707.78,A -85,B 0,C 180,E1 -6928.324,E2 -6928.324} C_VEL
LIN {X 0,Y 480.741,Z 708.398,A -85,B 0,C 180,E1 -6930,E2 -6930} C_VEL
LIN {X 0,Y 480.822,Z 707.808,A -85,B 0,C 180,E1 -6931.675,E2 -6931.675} C_VEL
LIN {X 0,Y 480.873,Z 706.05,A -85,B 0,C 180,E1 -6933.351,E2 -6933.351} C_VEL
LIN {X 0,Y 480.853,Z 703.096,A -85,B 0,C 180,E1 -6935.031,E2 -6935.031} C_VEL
LIN {X 0,Y 480.902,Z 698.882,A -85,B 0,C 180,E1 -6936.714,E2 -6936.714} C_VEL
LIN {X 0,Y 481.057,Z 693.298,A -85,B 0,C 180,E1 -6938.4,E2 -6938.4} C_VEL
LIN {X 0,Y 481.258,Z 686.19,A -85,B 0,C 180,E1 -6940.092,E2 -6940.092} C_VEL
LIN {X 0,Y 481.604,Z 678.596,A -85,B 0,C 180,E1 -6941.575,E2 -6941.575} C_VEL
LIN {X 0,Y 482.017,Z 669.439,A -85,B 0,C 180,E1 -6943.061,E2 -6943.061} C_VEL
LIN {X 0,Y 482.59,Z 658.419,A -85,B 0,C 180,E1 -6944.549,E2 -6944.549} C_VEL
LIN {X 0,Y 483.287,Z 647.095,A -85,B 0,C 180,E1 -6945.822,E2 -6945.822} C_VEL
LIN {X 0,Y 483.977,Z 634.673,A -85,B 0,C 180,E1 -6946.992,E2 -6946.992} C_VEL
LIN {X 0,Y 484.731,Z 620.986,A -85,B 0,C 180,E1 -6948.053,E2 -6948.053} C_VEL
LIN {X 0,Y 485.45,Z 607.553,A -85,B 0,C 180,E1 -6948.9,E2 -6948.9} C_VEL
LIN {X 0,Y 486.25,Z 592.38,A -85,B 0,C 180,E1 -6949.655,E2 -6949.655} C_VEL
LIN {X 0,Y 486.762,Z 577.068,A -85,B 0,C 180,E1 -6950.23,E2 -6950.23} C_VEL
LIN {X 0,Y 487.268,Z 560.916,A -85,B 0,C 180,E1 -6950.638,E2 -6950.638} C_VEL
LIN {X 0,Y 488.905,Z 417.97,A -85,B 0,C 180,E1 -6952.837,E2 -6952.837} C_VEL
LIN {X 0,Y 484.762,Z 394.773,A -85,B 0,C 180,E1 -6953.419,E2 -6953.419} C_VEL
LIN {X 0,Y 485.929,Z 370.536,A -85,B 0,C 180,E1 -6956.638,E2 -6956.638} C_VEL
LIN {X 0,Y 486.332,Z 359.204,A -85,B 0,C 180,E1 -6958.175,E2 -6958.175} C_VEL
LIN {X 0,Y 482.321,Z 342.774,A -85,B 0,C 180,E1 -6960.717,E2 -6960.717} C_VEL
LIN {X 0,Y 481.673,Z 340.112,A -85,B 0,C 180,E1 -6961.165,E2 -6961.165} C_VEL
LIN {X 0,Y 481.695,Z 340.108,A -85,B 0,C 180,E1 -6963.733,E2 -6963.733} C_VEL
LIN {X 0,Y 481.623,Z 340.118,A -85,B 0,C 180,E1 -6966.747,E2 -6966.747} C_VEL
LIN {X 0,Y 481.674,Z 340.107,A -85,B 0,C 180,E1 -6969.94,E2 -6969.94} C_VEL
LIN {X 0,Y 481.664,Z 340.115,A -85,B 0,C 180,E1 -6973.296,E2 -6973.296} C_VEL
LIN {X 0,Y 481.667,Z 340.109,A -85,B 0,C 180,E1 -6976.704,E2 -6976.704} C_VEL
LIN {X 0,Y 481.674,Z 340.106,A -85,B 0,C 180,E1 -6980.06,E2 -6980.06} C_VEL
LIN {X 0,Y 481.627,Z 340.119,A -85,B 0,C 180,E1 -6983.253,E2 -6983.253} C_VEL
LIN {X 0,Y 481.706,Z 340.102,A -85,B 0,C 180,E1 -6986.33,E2 -6986.33} C_VEL
LIN {X 0,Y 481.647,Z 340.113,A -85,B 0,C 180,E1 -6989.417,E2 -6989.417} C_VEL
LIN {X 0,Y 481.696,Z 340.103,A -85,B 0,C 180,E1 -6992.168,E2 -6992.168} C_VEL
LIN {X 0,Y 481.715,Z 340.108,A -85,B 0,C 180,E1 -6994.97,E2 -6994.97} C_VEL
LIN {X 0,Y 481.647,Z 340.11,A -85,B 0,C 180,E1 -6997.705,E2 -6997.705} C_VEL
LIN {X 0,Y 481.705,Z 340.103,A -85,B 0,C 180,E1 -7000.393,E2 -7000.393} C_VEL
LIN {X 0,Y 481.688,Z 340.113,A -85,B 0,C 180,E1 -7003.034,E2 -7003.034} C_VEL
LIN {X 0,Y 481.688,Z 340.105,A -85,B 0,C 180,E1 -7005.639,E2 -7005.639} C_VEL
LIN {X 0,Y 481.748,Z 340.097,A -85,B 0,C 180,E1 -7008.215,E2 -7008.215} C_VEL
LIN {X 0,Y 481.76,Z 340.096,A -85,B 0,C 180,E1 -7011.612,E2 -7011.612} C_VEL
LIN {X 0,Y 481.806,Z 340.09,A -85,B 0,C 180,E1 -7014.14,E2 -7014.14} C_VEL
LIN {X 0,Y 481.926,Z 340.076,A -85,B 0,C 180,E1 -7017.493,E2 -7017.493} C_VEL
LIN {X 0,Y 481.903,Z 340.085,A -85,B 0,C 180,E1 -7020.836,E2 -7020.836} C_VEL
LIN {X 0,Y 481.926,Z 340.078,A -85,B 0,C 180,E1 -7022.508,E2 -7022.508} C_VEL
LIN {X 0,Y 481.816,Z 340.088,A -85,B 0,C 180,E1 -7025.861,E2 -7025.861} C_VEL
LIN {X 0,Y 481.761,Z 340.097,A -85,B 0,C 180,E1 -7028.389,E2 -7028.389} C_VEL
LIN {X 0,Y 481.749,Z 340.096,A -85,B 0,C 180,E1 -7031.785,E2 -7031.785} C_VEL
LIN {X 0,Y 481.741,Z 340.1,A -85,B 0,C 180,E1 -7035.225,E2 -7035.225} C_VEL
LIN {X 0,Y 481.71,Z 340.109,A -85,B 0,C 180,E1 -7038.722,E2 -7038.722} C_VEL
LIN {X 0,Y 481.644,Z 340.111,A -85,B 0,C 180,E1 -7041.395,E2 -7041.395} C_VEL
LIN {X 0,Y 481.669,Z 340.107,A -85,B 0,C 180,E1 -7044.114,E2 -7044.114} C_VEL
LIN {X 0,Y 481.712,Z 340.104,A -85,B 0,C 180,E1 -7047.132,E2 -7047.132} C_VEL
LIN {X 0,Y 481.677,Z 340.105,A -85,B 0,C 180,E1 -7049.742,E2 -7049.742} C_VEL
LIN {X 0,Y 481.671,Z 340.115,A -85,B 0,C 180,E1 -7052.675,E2 -7052.675} C_VEL
LIN {X 0,Y 481.641,Z 340.11,A -85,B 0,C 180,E1 -7055.71,E2 -7055.71} C_VEL
LIN {X 0,Y 481.67,Z 340.111,A -85,B 0,C 180,E1 -7058.86,E2 -7058.86} C_VEL
LIN {X 0,Y 481.646,Z 340.11,A -85,B 0,C 180,E1 -7061.913,E2 -7061.913} C_VEL
LIN {X 0,Y 481.654,Z 340.115,A -85,B 0,C 180,E1 -7064.459,E2 -7064.459} C_VEL
LIN {X 0,Y 481.644,Z 340.11,A -85,B 0,C 180,E1 -7067.839,E2 -7067.839} C_VEL
LIN {X 0,Y 481.66,Z 340.114,A -85,B 0,C 180,E1 -7070.655,E2 -7070.655} C_VEL
LIN {X 0,Y 481.623,Z 340.112,A -85,B 0,C 180,E1 -7073.378,E2 -7073.378} C_VEL
LIN {X 0,Y 481.712,Z 340.107,A -85,B 0,C 180,E1 -7076.331,E2 -7076.331} C_VEL
LIN {X 0,Y 481.651,Z 340.108,A -85,B 0,C 180,E1 -7079.418,E2 -7079.418} C_VEL
LIN {X 0,Y 481.669,Z 340.111,A -85,B 0,C 180,E1 -7082.167,E2 -7082.167} C_VEL
LIN {X 0,Y 481.677,Z 340.107,A -85,B 0,C 180,E1 -7084.968,E2 -7084.968} C_VEL
LIN {X 0,Y 481.637,Z 340.111,A -85,B 0,C 180,E1 -7087.983,E2 -7087.983} C_VEL
LIN {X 0,Y 480.972,Z 340.198,A -85,B 0,C 180,E1 -7088.681,E2 -7088.681} C_VEL
LIN {X 0,Y 478.151,Z 340.546,A -85,B 0,C 180,E1 -7089.816,E2 -7089.816} C_VEL
LIN {X 0,Y 475.762,Z 340.846,A -85,B 0,C 180,E1 -7090.73,E2 -7090.73} C_VEL
LIN {X 0,Y 474.73,Z 340.971,A -85,B 0,C 180,E1 -7091.436,E2 -7091.436} C_VEL
LIN {X 0,Y 474.642,Z 340.982,A -85,B 0,C 180,E1 -7091.675,E2 -7091.675} C_VEL
LIN {X 0,Y 474.691,Z 340.982,A -85,B 0,C 180,E1 -7094.544,E2 -7094.544} C_VEL
LIN {X 0,Y 474.708,Z 340.978,A -85,B 0,C 180,E1 -7098.038,E2 -7098.038} C_VEL
LIN {X 0,Y 474.7,Z 340.975,A -85,B 0,C 180,E1 -7101.486,E2 -7101.486} C_VEL
LIN {X 0,Y 474.74,Z 340.974,A -85,B 0,C 180,E1 -7104.052,E2 -7104.052} C_VEL
LIN {X 0,Y 474.876,Z 340.953,A -85,B 0,C 180,E1 -7107.456,E2 -7107.456} C_VEL
LIN {X 0,Y 474.883,Z 340.956,A -85,B 0,C 180,E1 -7110,E2 -7110} C_VEL
LIN {X 0,Y 474.875,Z 340.957,A -85,B 0,C 180,E1 -7112.545,E2 -7112.545} C_VEL
LIN {X 0,Y 474.741,Z 340.974,A -85,B 0,C 180,E1 -7115.948,E2 -7115.948} C_VEL
LIN {X 0,Y 474.669,Z 340.982,A -85,B 0,C 180,E1 -7118.515,E2 -7118.515} C_VEL
LIN {X 0,Y 474.697,Z 340.982,A -85,B 0,C 180,E1 -7121.963,E2 -7121.963} C_VEL
LIN {X 0,Y 474.671,Z 341.157,A -85,B 0,C 180,E1 -7125.495,E2 -7125.495} C_VEL
LIN {X 0,Y 475.475,Z 344.885,A -85,B 0,C 180,E1 -7126.19,E2 -7126.19} C_VEL
LIN {X 0,Y 482.349,Z 362.118,A -85,B 0,C 180,E1 -7126.834,E2 -7126.834} C_VEL
LIN {X 0,Y 482.578,Z 365.905,A -85,B 0,C 180,E1 -7126.907,E2 -7126.907} C_VEL
LIN {X 0,Y 480.827,Z 509.305,A -85,B 0,C 180,E1 -7129.159,E2 -7129.159} C_VEL
LIN {X 0,Y 480.426,Z 524.902,A -85,B 0,C 180,E1 -7129.578,E2 -7129.578} C_VEL
LIN {X 0,Y 479.95,Z 538.987,A -85,B 0,C 180,E1 -7130.12,E2 -7130.12} C_VEL
LIN {X 0,Y 479.274,Z 554.079,A -85,B 0,C 180,E1 -7130.887,E2 -7130.887} C_VEL
LIN {X 0,Y 478.522,Z 568.271,A -85,B 0,C 180,E1 -7131.807,E2 -7131.807} C_VEL
LIN {X 0,Y 477.748,Z 581.109,A -85,B 0,C 180,E1 -7132.83,E2 -7132.83} C_VEL
LIN {X 0,Y 476.971,Z 593.223,A -85,B 0,C 180,E1 -7133.998,E2 -7133.998} C_VEL
LIN {X 0,Y 476.232,Z 604.779,A -85,B 0,C 180,E1 -7135.339,E2 -7135.339} C_VEL
LIN {X 0,Y 475.544,Z 615.208,A -85,B 0,C 180,E1 -7136.793,E2 -7136.793} C_VEL
LIN {X 0,Y 475.018,Z 623.965,A -85,B 0,C 180,E1 -7138.259,E2 -7138.259} C_VEL
LIN {X 0,Y 474.567,Z 631.355,A -85,B 0,C 180,E1 -7139.743,E2 -7139.743} C_VEL
LIN {X 0,Y 474.307,Z 637.525,A -85,B 0,C 180,E1 -7141.239,E2 -7141.239} C_VEL
LIN {X 0,Y 474.055,Z 642.689,A -85,B 0,C 180,E1 -7142.768,E2 -7142.768} C_VEL
LIN {X 0,Y 473.912,Z 646.766,A -85,B 0,C 180,E1 -7144.301,E2 -7144.301} C_VEL
LIN {X 0,Y 473.772,Z 648.969,A -85,B 0,C 180,E1 -7145.348,E2 -7145.348} C_VEL
LIN {X 0,Y 473.683,Z 651.161,A -85,B 0,C 180,E1 -7146.755,E2 -7146.755} C_VEL
LIN {X 0,Y 473.651,Z 652.859,A -85,B 0,C 180,E1 -7148.55,E2 -7148.55} C_VEL
LIN {X 0,Y 473.634,Z 653.278,A -85,B 0,C 180,E1 -7149.647,E2 -7149.647} C_VEL
LIN {X 0,Y 473.658,Z 653.221,A -85,B 0,C 180,E1 -7150.823,E2 -7150.823} C_VEL
LIN {X 0,Y 473.66,Z 652.529,A -85,B 0,C 180,E1 -7152.107,E2 -7152.107} C_VEL
LIN {X 0,Y 473.732,Z 651.196,A -85,B 0,C 180,E1 -7153.369,E2 -7153.369} C_VEL
LIN {X 0,Y 473.829,Z 649.309,A -85,B 0,C 180,E1 -7154.605,E2 -7154.605} C_VEL
LIN {X 0,Y 474.021,Z 644.923,A -85,B 0,C 180,E1 -7156.593,E2 -7156.593} C_VEL
LIN {X 0,Y 474.178,Z 640.174,A -85,B 0,C 180,E1 -7158.166,E2 -7158.166} C_VEL
LIN {X 0,Y 474.507,Z 633.677,A -85,B 0,C 180,E1 -7159.874,E2 -7159.874} C_VEL
LIN {X 0,Y 474.966,Z 625.6,A -85,B 0,C 180,E1 -7161.576,E2 -7161.576} C_VEL
LIN {X 0,Y 475.573,Z 616.353,A -85,B 0,C 180,E1 -7163.165,E2 -7163.165} C_VEL
LIN {X 0,Y 476.196,Z 606.433,A -85,B 0,C 180,E1 -7164.581,E2 -7164.581} C_VEL
LIN {X 0,Y 476.992,Z 594.899,A -85,B 0,C 180,E1 -7165.951,E2 -7165.951} C_VEL
LIN {X 0,Y 477.678,Z 583.28,A -85,B 0,C 180,E1 -7167.103,E2 -7167.103} C_VEL
LIN {X 0,Y 478.456,Z 570.251,A -85,B 0,C 180,E1 -7168.174,E2 -7168.174} C_VEL
LIN {X 0,Y 479.192,Z 557.916,A -85,B 0,C 180,E1 -7169.003,E2 -7169.003} C_VEL
LIN {X 0,Y 479.752,Z 544.829,A -85,B 0,C 180,E1 -7169.724,E2 -7169.724} C_VEL
LIN {X 0,Y 480.327,Z 530.621,A -85,B 0,C 180,E1 -7170.332,E2 -7170.332} C_VEL
LIN {X 0,Y 480.739,Z 515.774,A -85,B 0,C 180,E1 -7170.796,E2 -7170.796} C_VEL
LIN {X 0,Y 480.992,Z 500.035,A -85,B 0,C 180,E1 -7171.112,E2 -7171.112} C_VEL
LIN {X 0,Y 482.742,Z 363.123,A -85,B 0,C 180,E1 -7173.259,E2 -7173.259} C_VEL
LIN {X 0,Y 475.773,Z 345.985,A -85,B 0,C 180,E1 -7173.93,E2 -7173.93} C_VEL
LIN {X 0,Y 474.642,Z 340.989,A -85,B 0,C 180,E1 -7174.98,E2 -7174.98} C_VEL
LIN {X 0,Y 474.583,Z 340.993,A -85,B 0,C 180,E1 -7178.27,E2 -7178.27} C_VEL
LIN {X 0,Y 474.658,Z 340.983,A -85,B 0,C 180,E1 -7181.373,E2 -7181.373} C_VEL
LIN {X 0,Y 474.691,Z 340.979,A -85,B 0,C 180,E1 -7184.544,E2 -7184.544} C_VEL
LIN {X 0,Y 474.708,Z 340.98,A -85,B 0,C 180,E1 -7188.037,E2 -7188.037} C_VEL
LIN {X 0,Y 474.699,Z 340.981,A -85,B 0,C 180,E1 -7191.486,E2 -7191.486} C_VEL
LIN {X 0,Y 474.741,Z 340.974,A -85,B 0,C 180,E1 -7194.052,E2 -7194.052} C_VEL
LIN {X 0,Y 474.877,Z 340.958,A -85,B 0,C 180,E1 -7197.455,E2 -7197.455} C_VEL
LIN {X 0,Y 474.911,Z 340.953,A -85,B 0,C 180,E1 -7200,E2 -7200} C_VEL
LIN {X 0,Y 474.888,Z 340.952,A -85,B 0,C 180,E1 -7202.544,E2 -7202.544} C_VEL
LIN {X 0,Y 474.752,Z 340.972,A -85,B 0,C 180,E1 -7205.948,E2 -7205.948} C_VEL
LIN {X 0,Y 474.711,Z 340.975,A -85,B 0,C 180,E1 -7208.514,E2 -7208.514} C_VEL
LIN {X 0,Y 474.707,Z 340.975,A -85,B 0,C 180,E1 -7211.962,E2 -7211.962} C_VEL
LIN {X 0,Y 474.702,Z 340.978,A -85,B 0,C 180,E1 -7215.455,E2 -7215.455} C_VEL
LIN {X 0,Y 474.665,Z 340.982,A -85,B 0,C 180,E1 -7219.01,E2 -7219.01} C_VEL
LIN {X 0,Y 474.59,Z 340.991,A -85,B 0,C 180,E1 -7221.729,E2 -7221.729} C_VEL
LIN {X 0,Y 474.656,Z 340.98,A -85,B 0,C 180,E1 -7224.493,E2 -7224.493} C_VEL
LIN {X 0,Y 474.683,Z 340.982,A -85,B 0,C 180,E1 -7227.334,E2 -7227.334} C_VEL
LIN {X 0,Y 474.607,Z 340.986,A -85,B 0,C 180,E1 -7230.23,E2 -7230.23} C_VEL
LIN {X 0,Y 474.644,Z 340.99,A -85,B 0,C 180,E1 -7233.22,E2 -7233.22} C_VEL
LIN {X 0,Y 474.59,Z 340.992,A -85,B 0,C 180,E1 -7236.323,E2 -7236.323} C_VEL
LIN {X 0,Y 474.629,Z 340.987,A -85,B 0,C 180,E1 -7239.647,E2 -7239.647} C_VEL
LIN {X 0,Y 474.616,Z 340.992,A -85,B 0,C 180,E1 -7242.934,E2 -7242.934} C_VEL
LIN {X 0,Y 474.617,Z 340.987,A -85,B 0,C 180,E1 -7245.896,E2 -7245.896} C_VEL
LIN {X 0,Y 474.634,Z 340.991,A -85,B 0,C 180,E1 -7249.04,E2 -7249.04} C_VEL
LIN {X 0,Y 474.611,Z 340.99,A -85,B 0,C 180,E1 -7251.704,E2 -7251.704} C_VEL
LIN {X 0,Y 474.625,Z 340.99,A -85,B 0,C 180,E1 -7254.725,E2 -7254.725} C_VEL
LIN {X 0,Y 474.637,Z 340.988,A -85,B 0,C 180,E1 -7257.787,E2 -7257.787} C_VEL
LIN {X 0,Y 474.643,Z 341.096,A -85,B 0,C 180,E1 -7258.646,E2 -7258.646} C_VEL
LIN {X 0,Y 478.009,Z 354.55,A -85,B 0,C 180,E1 -7260.813,E2 -7260.813} C_VEL
LIN {X 0,Y 479.382,Z 361.086,A -85,B 0,C 180,E1 -7261.819,E2 -7261.819} C_VEL
LIN {X 0,Y 478.737,Z 376.009,A -85,B 0,C 180,E1 -7263.87,E2 -7263.87} C_VEL
LIN {X 0,Y 477.83,Z 393.284,A -85,B 0,C 180,E1 -7266.195,E2 -7266.195} C_VEL
LIN {X 0,Y 482.273,Z 418.32,A -85,B 0,C 180,E1 -7266.844,E2 -7266.844} C_VEL
LIN {X 0,Y 480.536,Z 560.744,A -85,B 0,C 180,E1 -7269.087,E2 -7269.087} C_VEL
LIN {X 0,Y 480.057,Z 576.529,A -85,B 0,C 180,E1 -7269.503,E2 -7269.503} C_VEL
LIN {X 0,Y 479.413,Z 591.543,A -85,B 0,C 180,E1 -7270.072,E2 -7270.072} C_VEL
LIN {X 0,Y 478.677,Z 606.406,A -85,B 0,C 180,E1 -7270.821,E2 -7270.821} C_VEL
LIN {X 0,Y 477.891,Z 619.902,A -85,B 0,C 180,E1 -7271.678,E2 -7271.678} C_VEL
LIN {X 0,Y 477.036,Z 633.656,A -85,B 0,C 180,E1 -7272.752,E2 -7272.752} C_VEL
LIN {X 0,Y 476.333,Z 646.158,A -85,B 0,C 180,E1 -7273.94,E2 -7273.94} C_VEL
LIN {X 0,Y 475.572,Z 657.559,A -85,B 0,C 180,E1 -7275.231,E2 -7275.231} C_VEL
LIN {X 0,Y 475.014,Z 668.659,A -85,B 0,C 180,E1 -7276.742,E2 -7276.742} C_VEL
LIN {X 0,Y 474.531,Z 677.881,A -85,B 0,C 180,E1 -7278.25,E2 -7278.25} C_VEL
LIN {X 0,Y 474.229,Z 685.536,A -85,B 0,C 180,E1 -7279.756,E2 -7279.756} C_VEL
LIN {X 0,Y 473.97,Z 692.69,A -85,B 0,C 180,E1 -7281.472,E2 -7281.472} C_VEL
LIN {X 0,Y 473.887,Z 698.325,A -85,B 0,C 180,E1 -7283.186,E2 -7283.186} C_VEL
LIN {X 0,Y 473.782,Z 702.584,A -85,B 0,C 180,E1 -7284.893,E2 -7284.893} C_VEL
LIN {X 0,Y 473.799,Z 705.579,A -85,B 0,C 180,E1 -7286.598,E2 -7286.598} C_VEL
LIN {X 0,Y 473.756,Z 707.369,A -85,B 0,C 180,E1 -7288.299,E2 -7288.299} C_VEL
LIN {X 0,Y 473.667,Z 707.99,A -85,B 0,C 180,E1 -7290,E2 -7290} C_VEL
LIN {X 0,Y 473.755,Z 707.403,A -85,B 0,C 180,E1 -7291.7,E2 -7291.7} C_VEL
LIN {X 0,Y 473.798,Z 705.645,A -85,B 0,C 180,E1 -7293.401,E2 -7293.401} C_VEL
LIN {X 0,Y 473.78,Z 702.689,A -85,B 0,C 180,E1 -7295.106,E2 -7295.106} C_VEL
LIN {X 0,Y 473.822,Z 698.471,A -85,B 0,C 180,E1 -7296.814,E2 -7296.814} C_VEL
LIN {X 0,Y 473.969,Z 692.882,A -85,B 0,C 180,E1 -7298.527,E2 -7298.527} C_VEL
LIN {X 0,Y 474.23,Z 685.771,A -85,B 0,C 180,E1 -7300.243,E2 -7300.243} C_VEL
LIN {X 0,Y 474.563,Z 678.169,A -85,B 0,C 180,E1 -7301.749,E2 -7301.749} C_VEL
LIN {X 0,Y 475.035,Z 669.005,A -85,B 0,C 180,E1 -7303.257,E2 -7303.257} C_VEL
LIN {X 0,Y 475.625,Z 657.967,A -85,B 0,C 180,E1 -7304.767,E2 -7304.767} C_VEL
LIN {X 0,Y 476.369,Z 646.63,A -85,B 0,C 180,E1 -7306.058,E2 -7306.058} C_VEL
LIN {X 0,Y 477.083,Z 634.189,A -85,B 0,C 180,E1 -7307.245,E2 -7307.245} C_VEL
LIN {X 0,Y 477.917,Z 620.481,A -85,B 0,C 180,E1 -7308.32,E2 -7308.32} C_VEL
LIN {X 0,Y 478.691,Z 607.032,A -85,B 0,C 180,E1 -7309.178,E2 -7309.178} C_VEL
LIN {X 0,Y 479.493,Z 592.224,A -85,B 0,C 180,E1 -7309.925,E2 -7309.925} C_VEL
LIN {X 0,Y 480.097,Z 576.386,A -85,B 0,C 180,E1 -7310.524,E2 -7310.524} C_VEL
LIN {X 0,Y 480.585,Z 561.536,A -85,B 0,C 180,E1 -7310.91,E2 -7310.91} C_VEL
LIN {X 0,Y 482.164,Z 427.765,A -85,B 0,C 180,E1 -7313.006,E2 -7313.006} C_VEL
LIN {X 0,Y 482.177,Z 417.837,A -85,B 0,C 180,E1 -7313.167,E2 -7313.167} C_VEL
LIN {X 0,Y 477.95,Z 394.352,A -85,B 0,C 180,E1 -7313.774,E2 -7313.774} C_VEL
LIN {X 0,Y 479.127,Z 371.441,A -85,B 0,C 180,E1 -7316.865,E2 -7316.865} C_VEL
LIN {X 0,Y 479.614,Z 361.596,A -85,B 0,C 180,E1 -7318.213,E2 -7318.213} C_VEL
LIN {X 0,Y 475.759,Z 345.405,A -85,B 0,C 180,E1 -7320.747,E2 -7320.747} C_VEL
LIN {X 0,Y 474.614,Z 340.992,A -85,B 0,C 180,E1 -7321.464,E2 -7321.464} C_VEL
LIN {X 0,Y 474.629,Z 340.987,A -85,B 0,C 180,E1 -7324.241,E2 -7324.241} C_VEL
LIN {X 0,Y 474.588,Z 340.997,A -85,B 0,C 180,E1 -7327.383,E2 -7327.383} C_VEL
LIN {X 0,Y 474.625,Z 340.987,A -85,B 0,C 180,E1 -7329.647,E2 -7329.647} C_VEL
LIN {X 0,Y 474.633,Z 340.987,A -85,B 0,C 180,E1 -7332.932,E2 -7332.932} C_VEL
LIN {X 0,Y 474.613,Z 340.986,A -85,B 0,C 180,E1 -7335.896,E2 -7335.896} C_VEL
LIN {X 0,Y 474.629,Z 340.99,A -85,B 0,C 180,E1 -7339.04,E2 -7339.04} C_VEL
LIN {X 0,Y 474.607,Z 340.988,A -85,B 0,C 180,E1 -7341.704,E2 -7341.704} C_VEL
LIN {X 0,Y 474.627,Z 340.986,A -85,B 0,C 180,E1 -7344.726,E2 -7344.726} C_VEL
LIN {X 0,Y 474.632,Z 340.984,A -85,B 0,C 180,E1 -7347.788,E2 -7347.788} C_VEL
LIN {X 0,Y 474.621,Z 340.99,A -85,B 0,C 180,E1 -7350.884,E2 -7350.884} C_VEL
LIN {X 0,Y 474.657,Z 340.982,A -85,B 0,C 180,E1 -7353.628,E2 -7353.628} C_VEL
LIN {X 0,Y 474.632,Z 340.986,A -85,B 0,C 180,E1 -7356.641,E2 -7356.641} C_VEL
LIN {X 0,Y 474.653,Z 340.98,A -85,B 0,C 180,E1 -7360.09,E2 -7360.09} C_VEL
LIN {X 0,Y 474.647,Z 340.986,A -85,B 0,C 180,E1 -7362.775,E2 -7362.775} C_VEL
LIN {X 0,Y 474.646,Z 340.984,A -85,B 0,C 180,E1 -7365.421,E2 -7365.421} C_VEL
LIN {X 0,Y 474.701,Z 340.974,A -85,B 0,C 180,E1 -7368.038,E2 -7368.038} C_VEL
LIN {X 0,Y 474.725,Z 340.973,A -85,B 0,C 180,E1 -7371.487,E2 -7371.487} C_VEL
LIN {X 0,Y 474.768,Z 340.966,A -85,B 0,C 180,E1 -7374.053,E2 -7374.053} C_VEL
LIN {X 0,Y 474.892,Z 340.952,A -85,B 0,C 180,E1 -7377.456,E2 -7377.456} C_VEL
LIN {X 0,Y 474.91,Z 340.948,A -85,B 0,C 180,E1 -7380,E2 -7380} C_VEL
LIN {X 0,Y 474.892,Z 340.954,A -85,B 0,C 180,E1 -7382.545,E2 -7382.545} C_VEL
LIN {X 0,Y 474.779,Z 340.965,A -85,B 0,C 180,E1 -7385.948,E2 -7385.948} C_VEL
LIN {X 0,Y 474.726,Z 340.975,A -85,B 0,C 180,E1 -7388.514,E2 -7388.514} C_VEL
LIN {X 0,Y 474.702,Z 340.974,A -85,B 0,C 180,E1 -7391.963,E2 -7391.963} C_VEL
LIN {X 0,Y 474.698,Z 340.976,A -85,B 0,C 180,E1 -7395.456,E2 -7395.456} C_VEL
LIN {X 0,Y 474.663,Z 340.984,A -85,B 0,C 180,E1 -7399.011,E2 -7399.011} C_VEL
